LIN {X 0,Y 354.801,Z 259.294,A -85,B 0,C 180,E1 -13349.685,E2 -13349.685} C_VEL
LIN {X 0,Y 354.812,Z 259.29,A -85,B 0,C 180,E1 -13353.685,E2 -13353.685} C_VEL
LIN {X 0,Y 354.795,Z 259.291,A -85,B 0,C 180,E1 -13356.461,E2 -13356.461} C_VEL
LIN {X 0,Y 354.823,Z 259.288,A -85,B 0,C 180,E1 -13359.425,E2 -13359.425} C_VEL
LIN {X 0,Y 354.787,Z 259.29,A -85,B 0,C 180,E1 -13362.869,E2 -13362.869} C_VEL
LIN {X 0,Y 354.791,Z 259.41,A -85,B 0,C 180,E1 -13364.212,E2 -13364.212} C_VEL
LIN {X 0,Y 355.557,Z 263.624,A -85,B 0,C 180,E1 -13367.776,E2 -13367.776} C_VEL
LIN {X 0,Y 356.179,Z 267.564,A -85,B 0,C 180,E1 -13370.847,E2 -13370.847} C_VEL
LIN {X 0,Y 356.609,Z 271.764,A -85,B 0,C 180,E1 -13373.905,E2 -13373.905} C_VEL
LIN {X 0,Y 356.289,Z 275.58,A -85,B 0,C 180,E1 -13376.475,E2 -13376.475} C_VEL
LIN {X 0,Y 355.724,Z 280.665,A -85,B 0,C 180,E1 -13379.749,E2 -13379.749} C_VEL
LIN {X 0,Y 355.068,Z 285.864,A -85,B 0,C 180,E1 -13382.964,E2 -13382.964} C_VEL
LIN {X 0,Y 354.552,Z 291.984,A -85,B 0,C 180,E1 -13386.645,E2 -13386.645} C_VEL
LIN {X 0,Y 354.356,Z 295.247,A -85,B 0,C 180,E1 -13388.455,E2 -13388.455} C_VEL
LIN {X 0,Y 357.769,Z 308.674,A -85,B 0,C 180,E1 -13389.219,E2 -13389.219} C_VEL
LIN {X 0,Y 360.089,Z 320.881,A -85,B 0,C 180,E1 -13390.079,E2 -13390.079} C_VEL
LIN {X 0,Y 361.243,Z 331.83,A -85,B 0,C 180,E1 -13390.982,E2 -13390.982} C_VEL
LIN {X 0,Y 360.677,Z 339.868,A -85,B 0,C 180,E1 -13391.688,E2 -13391.688} C_VEL
LIN {X 0,Y 359.136,Z 351.571,A -85,B 0,C 180,E1 -13392.931,E2 -13392.931} C_VEL
LIN {X 0,Y 357.813,Z 361.437,A -85,B 0,C 180,E1 -13394.249,E2 -13394.249} C_VEL
LIN {X 0,Y 356.726,Z 370.441,A -85,B 0,C 180,E1 -13395.744,E2 -13395.744} C_VEL
LIN {X 0,Y 355.47,Z 378.705,A -85,B 0,C 180,E1 -13397.439,E2 -13397.439} C_VEL
LIN {X 0,Y 354.633,Z 385.385,A -85,B 0,C 180,E1 -13399.149,E2 -13399.149} C_VEL
LIN {X 0,Y 353.992,Z 390.739,A -85,B 0,C 180,E1 -13400.861,E2 -13400.861} C_VEL
LIN {X 0,Y 353.547,Z 394.934,A -85,B 0,C 180,E1 -13402.576,E2 -13402.576} C_VEL
LIN {X 0,Y 353.314,Z 398.087,A -85,B 0,C 180,E1 -13404.292,E2 -13404.292} C_VEL
LIN {X 0,Y 353.266,Z 399.668,A -85,B 0,C 180,E1 -13405.436,E2 -13405.436} C_VEL
LIN {X 0,Y 353.22,Z 400.829,A -85,B 0,C 180,E1 -13406.578,E2 -13406.578} C_VEL
LIN {X 0,Y 353.204,Z 401.911,A -85,B 0,C 180,E1 -13408.86,E2 -13408.86} C_VEL
LIN {X 0,Y 353.264,Z 401.877,A -85,B 0,C 180,E1 -13410,E2 -13410} C_VEL
LIN {X 0,Y 353.223,Z 401.444,A -85,B 0,C 180,E1 -13411.14,E2 -13411.14} C_VEL
LIN {X 0,Y 353.226,Z 399.304,A -85,B 0,C 180,E1 -13413.422,E2 -13413.422} C_VEL
LIN {X 0,Y 353.258,Z 396.601,A -85,B 0,C 180,E1 -13415.136,E2 -13415.136} C_VEL
LIN {X 0,Y 353.419,Z 392.866,A -85,B 0,C 180,E1 -13416.852,E2 -13416.852} C_VEL
LIN {X 0,Y 353.702,Z 387.997,A -85,B 0,C 180,E1 -13418.57,E2 -13418.57} C_VEL
LIN {X 0,Y 354.198,Z 381.846,A -85,B 0,C 180,E1 -13420.287,E2 -13420.287} C_VEL
LIN {X 0,Y 354.851,Z 374.184,A -85,B 0,C 180,E1 -13422.002,E2 -13422.002} C_VEL
LIN {X 0,Y 355.604,Z 366.332,A -85,B 0,C 180,E1 -13423.428,E2 -13423.428} C_VEL
LIN {X 0,Y 356.485,Z 356.718,A -85,B 0,C 180,E1 -13424.85,E2 -13424.85} C_VEL
LIN {X 0,Y 357.37,Z 346.037,A -85,B 0,C 180,E1 -13426.127,E2 -13426.127} C_VEL
LIN {X 0,Y 358.522,Z 334.094,A -85,B 0,C 180,E1 -13427.247,E2 -13427.247} C_VEL
LIN {X 0,Y 358.749,Z 330.526,A -85,B 0,C 180,E1 -13427.529,E2 -13427.529} C_VEL
LIN {X 0,Y 357.34,Z 318.321,A -85,B 0,C 180,E1 -13428.423,E2 -13428.423} C_VEL
LIN {X 0,Y 355.4,Z 304.853,A -85,B 0,C 180,E1 -13429.164,E2 -13429.164} C_VEL
LIN {X 0,Y 353.852,Z 295.492,A -85,B 0,C 180,E1 -13429.544,E2 -13429.544} C_VEL
LIN {X 0,Y 354.18,Z 289.708,A -85,B 0,C 180,E1 -13432.764,E2 -13432.764} C_VEL
LIN {X 0,Y 354.551,Z 284.261,A -85,B 0,C 180,E1 -13435.854,E2 -13435.854} C_VEL
LIN {X 0,Y 355.08,Z 277.706,A -85,B 0,C 180,E1 -13439.657,E2 -13439.657} C_VEL
LIN {X 0,Y 355.598,Z 272.227,A -85,B 0,C 180,E1 -13442.922,E2 -13442.922} C_VEL
LIN {X 0,Y 355.985,Z 267.281,A -85,B 0,C 180,E1 -13445.957,E2 -13445.957} C_VEL
LIN {X 0,Y 355.526,Z 263.384,A -85,B 0,C 180,E1 -13448.511,E2 -13448.511} C_VEL
LIN {X 0,Y 354.84,Z 259.286,A -85,B 0,C 180,E1 -13451.394,E2 -13451.394} C_VEL
LIN {X 0,Y 354.743,Z 259.295,A -85,B 0,C 180,E1 -13455.496,E2 -13455.496} C_VEL
LIN {X 0,Y 354.76,Z 259.294,A -85,B 0,C 180,E1 -13459.174,E2 -13459.174} C_VEL
LIN {X 0,Y 354.796,Z 259.29,A -85,B 0,C 180,E1 -13462.403,E2 -13462.403} C_VEL
LIN {X 0,Y 354.805,Z 259.29,A -85,B 0,C 180,E1 -13464.939,E2 -13464.939} C_VEL
LIN {X 0,Y 354.79,Z 259.292,A -85,B 0,C 180,E1 -13468.404,E2 -13468.404} C_VEL
LIN {X 0,Y 354.796,Z 259.287,A -85,B 0,C 180,E1 -13471.613,E2 -13471.613} C_VEL
LIN {X 0,Y 354.83,Z 259.283,A -85,B 0,C 180,E1 -13475.656,E2 -13475.656} C_VEL
LIN {X 0,Y 354.821,Z 259.285,A -85,B 0,C 180,E1 -13479.112,E2 -13479.112} C_VEL
LIN {X 0,Y 354.893,Z 259.277,A -85,B 0,C 180,E1 -13482.718,E2 -13482.718} C_VEL
LIN {X 0,Y 354.946,Z 259.274,A -85,B 0,C 180,E1 -13486.254,E2 -13486.254} C_VEL
LIN {X 0,Y 354.971,Z 259.268,A -85,B 0,C 180,E1 -13489.734,E2 -13489.734} C_VEL
LIN {X 0,Y 355.119,Z 259.247,A -85,B 0,C 180,E1 -13493.179,E2 -13493.179} C_VEL
LIN {X 0,Y 355.237,Z 259.236,A -85,B 0,C 180,E1 -13497.731,E2 -13497.731} C_VEL
LIN {X 0,Y 355.391,Z 259.218,A -85,B 0,C 180,E1 -13499.999,E2 -13499.999} C_VEL
LIN {X 0,Y 355.238,Z 259.234,A -85,B 0,C 180,E1 -13502.266,E2 -13502.266} C_VEL
LIN {X 0,Y 355.13,Z 259.246,A -85,B 0,C 180,E1 -13506.818,E2 -13506.818} C_VEL
LIN {X 0,Y 355.007,Z 259.262,A -85,B 0,C 180,E1 -13509.111,E2 -13509.111} C_VEL
LIN {X 0,Y 354.912,Z 259.273,A -85,B 0,C 180,E1 -13512.58,E2 -13512.58} C_VEL
LIN {X 0,Y 354.879,Z 259.278,A -85,B 0,C 180,E1 -13516.095,E2 -13516.095} C_VEL
LIN {X 0,Y 354.891,Z 259.275,A -85,B 0,C 180,E1 -13518.471,E2 -13518.471} C_VEL
LIN {X 0,Y 354.824,Z 259.284,A -85,B 0,C 180,E1 -13522.105,E2 -13522.105} C_VEL
LIN {X 0,Y 354.889,Z 259.277,A -85,B 0,C 180,E1 -13525.826,E2 -13525.826} C_VEL
LIN {X 0,Y 354.844,Z 259.283,A -85,B 0,C 180,E1 -13529.678,E2 -13529.678} C_VEL
LIN {X 0,Y 354.795,Z 259.288,A -85,B 0,C 180,E1 -13533.701,E2 -13533.701} C_VEL
LIN {X 0,Y 354.788,Z 259.289,A -85,B 0,C 180,E1 -13536.459,E2 -13536.459} C_VEL
LIN {X 0,Y 354.813,Z 259.287,A -85,B 0,C 180,E1 -13539.423,E2 -13539.423} C_VEL
LIN {X 0,Y 354.823,Z 259.29,A -85,B 0,C 180,E1 -13542.875,E2 -13542.875} C_VEL
LIN {X 0,Y 354.773,Z 259.29,A -85,B 0,C 180,E1 -13546.106,E2 -13546.106} C_VEL
LIN {X 0,Y 354.777,Z 259.291,A -85,B 0,C 180,E1 -13549.179,E2 -13549.179} C_VEL
LIN {X 0,Y 354.8,Z 259.29,A -85,B 0,C 180,E1 -13552.401,E2 -13552.401} C_VEL
LIN {X 0,Y 354.8,Z 259.289,A -85,B 0,C 180,E1 -13554.94,E2 -13554.94} C_VEL
LIN {X 0,Y 354.782,Z 259.294,A -85,B 0,C 180,E1 -13558.405,E2 -13558.405} C_VEL
LIN {X 0,Y 354.825,Z 259.284,A -85,B 0,C 180,E1 -13561.617,E2 -13561.617} C_VEL
LIN {X 0,Y 354.816,Z 259.288,A -85,B 0,C 180,E1 -13564.167,E2 -13564.167} C_VEL
LIN {X 0,Y 354.703,Z 259.301,A -85,B 0,C 180,E1 -13566.655,E2 -13566.655} C_VEL
LIN {X 0,Y 354.621,Z 259.436,A -85,B 0,C 180,E1 -13568.344,E2 -13568.344} C_VEL
LIN {X 0,Y 354.458,Z 263.774,A -85,B 0,C 180,E1 -13572.117,E2 -13572.117} C_VEL
LIN {X 0,Y 354.257,Z 268.889,A -85,B 0,C 180,E1 -13576.425,E2 -13576.425} C_VEL
LIN {X 0,Y 354.011,Z 274.308,A -85,B 0,C 180,E1 -13580.862,E2 -13580.862} C_VEL
LIN {X 0,Y 354.001,Z 277.677,A -85,B 0,C 180,E1 -13583.549,E2 -13583.549} C_VEL
LIN {X 0,Y 356.74,Z 290.857,A -85,B 0,C 180,E1 -13584.182,E2 -13584.182} C_VEL
LIN {X 0,Y 358.805,Z 303.884,A -85,B 0,C 180,E1 -13585.014,E2 -13585.014} C_VEL
LIN {X 0,Y 359.321,Z 308.615,A -85,B 0,C 180,E1 -13585.372,E2 -13585.372} C_VEL
LIN {X 0,Y 358.466,Z 320.435,A -85,B 0,C 180,E1 -13586.347,E2 -13586.347} C_VEL
LIN {X 0,Y 357.382,Z 332.207,A -85,B 0,C 180,E1 -13587.605,E2 -13587.605} C_VEL
LIN {X 0,Y 356.509,Z 341.682,A -85,B 0,C 180,E1 -13588.87,E2 -13588.87} C_VEL
LIN {X 0,Y 355.705,Z 350.333,A -85,B 0,C 180,E1 -13590.283,E2 -13590.283} C_VEL
LIN {X 0,Y 354.784,Z 358.758,A -85,B 0,C 180,E1 -13591.987,E2 -13591.987} C_VEL
LIN {X 0,Y 354.232,Z 365.515,A -85,B 0,C 180,E1 -13593.697,E2 -13593.697} C_VEL
LIN {X 0,Y 353.784,Z 371.732,A -85,B 0,C 180,E1 -13595.7,E2 -13595.7} C_VEL
LIN {X 0,Y 353.482,Z 375.785,A -85,B 0,C 180,E1 -13597.425,E2 -13597.425} C_VEL
LIN {X 0,Y 353.222,Z 378.791,A -85,B 0,C 180,E1 -13599.159,E2 -13599.159} C_VEL
LIN {X 0,Y 353.115,Z 380.238,A -85,B 0,C 180,E1 -13600.319,E2 -13600.319} C_VEL
LIN {X 0,Y 353.117,Z 381.259,A -85,B 0,C 180,E1 -13601.48,E2 -13601.48} C_VEL
LIN {X 0,Y 353.144,Z 381.957,A -85,B 0,C 180,E1 -13602.806,E2 -13602.806} C_VEL
LIN {X 0,Y 353.098,Z 381.895,A -85,B 0,C 180,E1 -13604.995,E2 -13604.995} C_VEL
LIN {X 0,Y 353.224,Z 381.265,A -85,B 0,C 180,E1 -13606.173,E2 -13606.173} C_VEL
LIN {X 0,Y 353.36,Z 380.231,A -85,B 0,C 180,E1 -13607.357,E2 -13607.357} C_VEL
LIN {X 0,Y 353.527,Z 378.734,A -85,B 0,C 180,E1 -13608.546,E2 -13608.546} C_VEL
LIN {X 0,Y 353.964,Z 375.623,A -85,B 0,C 180,E1 -13610.332,E2 -13610.332} C_VEL
LIN {X 0,Y 354.54,Z 371.367,A -85,B 0,C 180,E1 -13612.125,E2 -13612.125} C_VEL
LIN {X 0,Y 355.463,Z 364.784,A -85,B 0,C 180,E1 -13614.22,E2 -13614.22} C_VEL
LIN {X 0,Y 356.534,Z 357.492,A -85,B 0,C 180,E1 -13616.013,E2 -13616.013} C_VEL
LIN {X 0,Y 357.608,Z 350.251,A -85,B 0,C 180,E1 -13617.452,E2 -13617.452} C_VEL
LIN {X 0,Y 358.904,Z 340.748,A -85,B 0,C 180,E1 -13618.989,E2 -13618.989} C_VEL
LIN {X 0,Y 360.219,Z 330.531,A -85,B 0,C 180,E1 -13620.319,E2 -13620.319} C_VEL
LIN {X 0,Y 361.445,Z 319.694,A -85,B 0,C 180,E1 -13621.443,E2 -13621.443} C_VEL
LIN {X 0,Y 362.367,Z 310.873,A -85,B 0,C 180,E1 -13622.179,E2 -13622.179} C_VEL
LIN {X 0,Y 360.465,Z 300.228,A -85,B 0,C 180,E1 -13623.086,E2 -13623.086} C_VEL
LIN {X 0,Y 356.959,Z 287.408,A -85,B 0,C 180,E1 -13624.031,E2 -13624.031} C_VEL
LIN {X 0,Y 354.026,Z 278.062,A -85,B 0,C 180,E1 -13624.629,E2 -13624.629} C_VEL
LIN {X 0,Y 354.261,Z 274.211,A -85,B 0,C 180,E1 -13627.95,E2 -13627.95} C_VEL
LIN {X 0,Y 354.295,Z 273.377,A -85,B 0,C 180,E1 -13628.691,E2 -13628.691} C_VEL
LIN {X 0,Y 353.72,Z 272.417,A -85,B 0,C 180,E1 -13629.629,E2 -13629.629} C_VEL
LIN {X 0,Y 351.022,Z 271.112,A -85,B 0,C 180,E1 -13631.165,E2 -13631.165} C_VEL
LIN {X 0,Y 348.724,Z 270.103,A -85,B 0,C 180,E1 -13632.409,E2 -13632.409} C_VEL
LIN {X 0,Y 347.77,Z 269.229,A -85,B 0,C 180,E1 -13633.367,E2 -13633.367} C_VEL
LIN {X 0,Y 347.711,Z 268.9,A -85,B 0,C 180,E1 -13633.689,E2 -13633.689} C_VEL
LIN {X 0,Y 347.998,Z 265.854,A -85,B 0,C 180,E1 -13636.637,E2 -13636.637} C_VEL
LIN {X 0,Y 348.017,Z 262.805,A -85,B 0,C 180,E1 -13639.745,E2 -13639.745} C_VEL
LIN {X 0,Y 347.754,Z 260.169,A -85,B 0,C 180,E1 -13642.68,E2 -13642.68} C_VEL
LIN {X 0,Y 347.737,Z 260.175,A -85,B 0,C 180,E1 -13645.957,E2 -13645.957} C_VEL
LIN {X 0,Y 347.753,Z 260.169,A -85,B 0,C 180,E1 -13649.654,E2 -13649.654} C_VEL
LIN {X 0,Y 347.841,Z 260.156,A -85,B 0,C 180,E1 -13652.745,E2 -13652.745} C_VEL
LIN {X 0,Y 347.789,Z 260.166,A -85,B 0,C 180,E1 -13656.164,E2 -13656.164} C_VEL
LIN {X 0,Y 347.826,Z 260.157,A -85,B 0,C 180,E1 -13659.912,E2 -13659.912} C_VEL
LIN {X 0,Y 347.857,Z 260.152,A -85,B 0,C 180,E1 -13662.36,E2 -13662.36} C_VEL
LIN {X 0,Y 347.888,Z 260.149,A -85,B 0,C 180,E1 -13665.972,E2 -13665.972} C_VEL
LIN {X 0,Y 347.919,Z 260.148,A -85,B 0,C 180,E1 -13669.527,E2 -13669.527} C_VEL
LIN {X 0,Y 348.082,Z 260.128,A -85,B 0,C 180,E1 -13673.043,E2 -13673.043} C_VEL
LIN {X 0,Y 348.2,Z 260.112,A -85,B 0,C 180,E1 -13677.688,E2 -13677.688} C_VEL
LIN {X 0,Y 348.315,Z 260.096,A -85,B 0,C 180,E1 -13680.001,E2 -13680.001} C_VEL
LIN {X 0,Y 348.2,Z 260.113,A -85,B 0,C 180,E1 -13682.315,E2 -13682.315} C_VEL
LIN {X 0,Y 348.097,Z 260.125,A -85,B 0,C 180,E1 -13686.959,E2 -13686.959} C_VEL
LIN {X 0,Y 347.922,Z 260.147,A -85,B 0,C 180,E1 -13690.476,E2 -13690.476} C_VEL
LIN {X 0,Y 347.893,Z 260.153,A -85,B 0,C 180,E1 -13694.151,E2 -13694.151} C_VEL
LIN {X 0,Y 347.887,Z 260.155,A -85,B 0,C 180,E1 -13698.292,E2 -13698.292} C_VEL
LIN {X 0,Y 347.784,Z 260.17,A -85,B 0,C 180,E1 -13701.636,E2 -13701.636} C_VEL
LIN {X 0,Y 347.795,Z 260.168,A -85,B 0,C 180,E1 -13705.111,E2 -13705.111} C_VEL
LIN {X 0,Y 347.756,Z 260.172,A -85,B 0,C 180,E1 -13707.7,E2 -13707.7} C_VEL
LIN {X 0,Y 347.738,Z 260.174,A -85,B 0,C 180,E1 -13710.35,E2 -13710.35} C_VEL
LIN {X 0,Y 347.746,Z 260.171,A -85,B 0,C 180,E1 -13714.045,E2 -13714.045} C_VEL
LIN {X 0,Y 347.759,Z 260.167,A -85,B 0,C 180,E1 -13717.322,E2 -13717.322} C_VEL
LIN {X 0,Y 347.731,Z 260.165,A -85,B 0,C 180,E1 -13720.299,E2 -13720.299} C_VEL
LIN {X 0,Y 347.729,Z 260.194,A -85,B 0,C 180,E1 -13723.608,E2 -13723.608} C_VEL
LIN {X 0,Y 348.362,Z 263.721,A -85,B 0,C 180,E1 -13726.693,E2 -13726.693} C_VEL
LIN {X 0,Y 349.028,Z 267.661,A -85,B 0,C 180,E1 -13729.923,E2 -13729.923} C_VEL
LIN {X 0,Y 349.554,Z 271.573,A -85,B 0,C 180,E1 -13732.904,E2 -13732.904} C_VEL
LIN {X 0,Y 349.45,Z 275.595,A -85,B 0,C 180,E1 -13735.729,E2 -13735.729} C_VEL
LIN {X 0,Y 348.692,Z 281.673,A -85,B 0,C 180,E1 -13739.744,E2 -13739.744} C_VEL
LIN {X 0,Y 347.895,Z 287.826,A -85,B 0,C 180,E1 -13743.614,E2 -13743.614} C_VEL
LIN {X 0,Y 347.477,Z 292.973,A -85,B 0,C 180,E1 -13746.772,E2 -13746.772} C_VEL
LIN {X 0,Y 347.353,Z 294.823,A -85,B 0,C 180,E1 -13747.889,E2 -13747.889} C_VEL
LIN {X 0,Y 350.974,Z 309.105,A -85,B 0,C 180,E1 -13748.744,E2 -13748.744} C_VEL
LIN {X 0,Y 353.166,Z 320.098,A -85,B 0,C 180,E1 -13749.547,E2 -13749.547} C_VEL
LIN {X 0,Y 354.42,Z 330.812,A -85,B 0,C 180,E1 -13750.451,E2 -13750.451} C_VEL
LIN {X 0,Y 354.501,Z 335.805,A -85,B 0,C 180,E1 -13750.907,E2 -13750.907} C_VEL
LIN {X 0,Y 353.103,Z 347.135,A -85,B 0,C 180,E1 -13752.031,E2 -13752.031} C_VEL
LIN {X 0,Y 351.582,Z 357.393,A -85,B 0,C 180,E1 -13753.301,E2 -13753.301} C_VEL
LIN {X 0,Y 350.502,Z 365.948,A -85,B 0,C 180,E1 -13754.621,E2 -13754.621} C_VEL
LIN {X 0,Y 349.196,Z 374.926,A -85,B 0,C 180,E1 -13756.321,E2 -13756.321} C_VEL
LIN {X 0,Y 348.021,Z 382.301,A -85,B 0,C 180,E1 -13758.054,E2 -13758.054} C_VEL
LIN {X 0,Y 347.144,Z 389.122,A -85,B 0,C 180,E1 -13760.091,E2 -13760.091} C_VEL
LIN {X 0,Y 346.647,Z 393.641,A -85,B 0,C 180,E1 -13761.841,E2 -13761.841} C_VEL
LIN {X 0,Y 346.246,Z 397.795,A -85,B 0,C 180,E1 -13764.044,E2 -13764.044} C_VEL
LIN {X 0,Y 346.166,Z 399.556,A -85,B 0,C 180,E1 -13765.342,E2 -13765.342} C_VEL
LIN {X 0,Y 346.143,Z 400.678,A -85,B 0,C 180,E1 -13766.508,E2 -13766.508} C_VEL
LIN {X 0,Y 346.105,Z 401.72,A -85,B 0,C 180,E1 -13768.837,E2 -13768.837} C_VEL
LIN {X 0,Y 346.166,Z 401.667,A -85,B 0,C 180,E1 -13770,E2 -13770} C_VEL
LIN {X 0,Y 346.124,Z 401.198,A -85,B 0,C 180,E1 -13771.163,E2 -13771.163} C_VEL
LIN {X 0,Y 346.15,Z 399.018,A -85,B 0,C 180,E1 -13773.492,E2 -13773.492} C_VEL
LIN {X 0,Y 346.189,Z 395.828,A -85,B 0,C 180,E1 -13775.483,E2 -13775.483} C_VEL
LIN {X 0,Y 346.44,Z 390.998,A -85,B 0,C 180,E1 -13777.577,E2 -13777.577} C_VEL
LIN {X 0,Y 346.861,Z 384.643,A -85,B 0,C 180,E1 -13779.623,E2 -13779.623} C_VEL
LIN {X 0,Y 347.423,Z 377.709,A -85,B 0,C 180,E1 -13781.375,E2 -13781.375} C_VEL
LIN {X 0,Y 348.379,Z 369.03,A -85,B 0,C 180,E1 -13783.117,E2 -13783.117} C_VEL
LIN {X 0,Y 349.301,Z 358.868,A -85,B 0,C 180,E1 -13784.752,E2 -13784.752} C_VEL
LIN {X 0,Y 350.15,Z 349.327,A -85,B 0,C 180,E1 -13785.99,E2 -13785.99} C_VEL
LIN {X 0,Y 351.042,Z 339.51,A -85,B 0,C 180,E1 -13787.025,E2 -13787.025} C_VEL
LIN {X 0,Y 351.795,Z 331.299,A -85,B 0,C 180,E1 -13787.73,E2 -13787.73} C_VEL
LIN {X 0,Y 350.483,Z 319.676,A -85,B 0,C 180,E1 -13788.625,E2 -13788.625} C_VEL
LIN {X 0,Y 348.643,Z 306.367,A -85,B 0,C 180,E1 -13789.404,E2 -13789.404} C_VEL
LIN {X 0,Y 346.777,Z 295.257,A -85,B 0,C 180,E1 -13789.882,E2 -13789.882} C_VEL
LIN {X 0,Y 347.155,Z 289.384,A -85,B 0,C 180,E1 -13793.251,E2 -13793.251} C_VEL
LIN {X 0,Y 347.668,Z 282.622,A -85,B 0,C 180,E1 -13797.194,E2 -13797.194} C_VEL
LIN {X 0,Y 348.239,Z 276.307,A -85,B 0,C 180,E1 -13800.972,E2 -13800.972} C_VEL
LIN {X 0,Y 348.803,Z 270.824,A -85,B 0,C 180,E1 -13804.344,E2 -13804.344} C_VEL
LIN {X 0,Y 348.947,Z 267.706,A -85,B 0,C 180,E1 -13806.328,E2 -13806.328} C_VEL
LIN {X 0,Y 348.458,Z 264.187,A -85,B 0,C 180,E1 -13808.698,E2 -13808.698} C_VEL
LIN {X 0,Y 347.785,Z 260.165,A -85,B 0,C 180,E1 -13811.608,E2 -13811.608} C_VEL
LIN {X 0,Y 347.69,Z 260.177,A -85,B 0,C 180,E1 -13815.028,E2 -13815.028} C_VEL
LIN {X 0,Y 347.704,Z 260.172,A -85,B 0,C 180,E1 -13818.404,E2 -13818.404} C_VEL
LIN {X 0,Y 347.759,Z 260.164,A -85,B 0,C 180,E1 -13822.013,E2 -13822.013} C_VEL
LIN {X 0,Y 347.74,Z 260.166,A -85,B 0,C 180,E1 -13825.534,E2 -13825.534} C_VEL
LIN {X 0,Y 347.742,Z 260.168,A -85,B 0,C 180,E1 -13828.299,E2 -13828.299} C_VEL
LIN {X 0,Y 347.742,Z 260.168,A -85,B 0,C 180,E1 -13830.983,E2 -13830.983} C_VEL
LIN {X 0,Y 347.744,Z 260.165,A -85,B 0,C 180,E1 -13833.599,E2 -13833.599} C_VEL
LIN {X 0,Y 347.762,Z 260.166,A -85,B 0,C 180,E1 -13836.159,E2 -13836.159} C_VEL
LIN {X 0,Y 347.8,Z 260.16,A -85,B 0,C 180,E1 -13839.907,E2 -13839.907} C_VEL
LIN {X 0,Y 347.861,Z 260.156,A -85,B 0,C 180,E1 -13842.358,E2 -13842.358} C_VEL
LIN {X 0,Y 347.893,Z 260.15,A -85,B 0,C 180,E1 -13845.969,E2 -13845.969} C_VEL
LIN {X 0,Y 347.922,Z 260.144,A -85,B 0,C 180,E1 -13849.524,E2 -13849.524} C_VEL
LIN {X 0,Y 348.085,Z 260.123,A -85,B 0,C 180,E1 -13853.041,E2 -13853.041} C_VEL
LIN {X 0,Y 348.2,Z 260.112,A -85,B 0,C 180,E1 -13857.685,E2 -13857.685} C_VEL
LIN {X 0,Y 348.361,Z 260.094,A -85,B 0,C 180,E1 -13859.999,E2 -13859.999} C_VEL
LIN {X 0,Y 348.201,Z 260.11,A -85,B 0,C 180,E1 -13862.312,E2 -13862.312} C_VEL
LIN {X 0,Y 348.098,Z 260.122,A -85,B 0,C 180,E1 -13866.956,E2 -13866.956} C_VEL
LIN {X 0,Y 347.959,Z 260.141,A -85,B 0,C 180,E1 -13869.297,E2 -13869.297} C_VEL
LIN {X 0,Y 347.881,Z 260.149,A -85,B 0,C 180,E1 -13872.838,E2 -13872.838} C_VEL
LIN {X 0,Y 347.829,Z 260.155,A -85,B 0,C 180,E1 -13876.43,E2 -13876.43} C_VEL
LIN {X 0,Y 347.841,Z 260.154,A -85,B 0,C 180,E1 -13878.859,E2 -13878.859} C_VEL
LIN {X 0,Y 347.764,Z 260.163,A -85,B 0,C 180,E1 -13882.578,E2 -13882.578} C_VEL
LIN {X 0,Y 347.802,Z 260.162,A -85,B 0,C 180,E1 -13885.107,E2 -13885.107} C_VEL
LIN {X 0,Y 347.802,Z 260.16,A -85,B 0,C 180,E1 -13887.693,E2 -13887.693} C_VEL
LIN {X 0,Y 347.754,Z 260.164,A -85,B 0,C 180,E1 -13890.346,E2 -13890.346} C_VEL
LIN {X 0,Y 347.733,Z 260.168,A -85,B 0,C 180,E1 -13894.463,E2 -13894.463} C_VEL
LIN {X 0,Y 347.765,Z 260.163,A -85,B 0,C 180,E1 -13897.988,E2 -13897.988} C_VEL
LIN {X 0,Y 347.773,Z 260.162,A -85,B 0,C 180,E1 -13901.608,E2 -13901.608} C_VEL
LIN {X 0,Y 347.785,Z 260.164,A -85,B 0,C 180,E1 -13905.011,E2 -13905.011} C_VEL
LIN {X 0,Y 347.739,Z 260.168,A -85,B 0,C 180,E1 -13908.397,E2 -13908.397} C_VEL
LIN {X 0,Y 347.765,Z 260.163,A -85,B 0,C 180,E1 -13912.01,E2 -13912.01} C_VEL
LIN {X 0,Y 347.733,Z 260.167,A -85,B 0,C 180,E1 -13915.536,E2 -13915.536} C_VEL
LIN {X 0,Y 347.733,Z 260.17,A -85,B 0,C 180,E1 -13918.3,E2 -13918.3} C_VEL
LIN {X 0,Y 347.763,Z 260.164,A -85,B 0,C 180,E1 -13920.987,E2 -13920.987} C_VEL
LIN {X 0,Y 347.775,Z 260.162,A -85,B 0,C 180,E1 -13923.604,E2 -13923.604} C_VEL
LIN {X 0,Y 347.686,Z 260.177,A -85,B 0,C 180,E1 -13926.155,E2 -13926.155} C_VEL
LIN {X 0,Y 347.579,Z 260.275,A -85,B 0,C 180,E1 -13928.297,E2 -13928.297} C_VEL
LIN {X 0,Y 347.387,Z 264.853,A -85,B 0,C 180,E1 -13932.334,E2 -13932.334} C_VEL
LIN {X 0,Y 347.194,Z 269.486,A -85,B 0,C 180,E1 -13936.311,E2 -13936.311} C_VEL
LIN {X 0,Y 346.957,Z 274.754,A -85,B 0,C 180,E1 -13940.674,E2 -13940.674} C_VEL
LIN {X 0,Y 346.953,Z 277.847,A -85,B 0,C 180,E1 -13943.211,E2 -13943.211} C_VEL
LIN {X 0,Y 349.868,Z 291.864,A -85,B 0,C 180,E1 -13943.914,E2 -13943.914} C_VEL
LIN {X 0,Y 351.753,Z 303.801,A -85,B 0,C 180,E1 -13944.698,E2 -13944.698} C_VEL
LIN {X 0,Y 352.418,Z 309.462,A -85,B 0,C 180,E1 -13945.138,E2 -13945.138} C_VEL
LIN {X 0,Y 351.521,Z 321.106,A -85,B 0,C 180,E1 -13946.131,E2 -13946.131} C_VEL
LIN {X 0,Y 350.421,Z 332.79,A -85,B 0,C 180,E1 -13947.414,E2 -13947.414} C_VEL
LIN {X 0,Y 349.646,Z 341.22,A -85,B 0,C 180,E1 -13948.56,E2 -13948.56} C_VEL
LIN {X 0,Y 348.756,Z 349.989,A -85,B 0,C 180,E1 -13950,E2 -13950} C_VEL
LIN {X 0,Y 347.79,Z 358.545,A -85,B 0,C 180,E1 -13951.737,E2 -13951.737} C_VEL
LIN {X 0,Y 347.216,Z 365.376,A -85,B 0,C 180,E1 -13953.481,E2 -13953.481} C_VEL
LIN {X 0,Y 346.773,Z 370.853,A -85,B 0,C 180,E1 -13955.233,E2 -13955.233} C_VEL
LIN {X 0,Y 346.473,Z 375.149,A -85,B 0,C 180,E1 -13956.99,E2 -13956.99} C_VEL
LIN {X 0,Y 346.286,Z 377.434,A -85,B 0,C 180,E1 -13958.167,E2 -13958.167} C_VEL
LIN {X 0,Y 346.114,Z 379.258,A -85,B 0,C 180,E1 -13959.348,E2 -13959.348} C_VEL
LIN {X 0,Y 346.022,Z 380.628,A -85,B 0,C 180,E1 -13960.532,E2 -13960.532} C_VEL
LIN {X 0,Y 346.015,Z 381.597,A -85,B 0,C 180,E1 -13961.719,E2 -13961.719} C_VEL
LIN {X 0,Y 346.04,Z 382.17,A -85,B 0,C 180,E1 -13962.909,E2 -13962.909} C_VEL
LIN {X 0,Y 346.016,Z 382.298,A -85,B 0,C 180,E1 -13964.107,E2 -13964.107} C_VEL
LIN {X 0,Y 346.023,Z 382.016,A -85,B 0,C 180,E1 -13965.31,E2 -13965.31} C_VEL
LIN {X 0,Y 346.299,Z 380.467,A -85,B 0,C 180,E1 -13967.482,E2 -13967.482} C_VEL
LIN {X 0,Y 346.664,Z 377.696,A -85,B 0,C 180,E1 -13969.542,E2 -13969.542} C_VEL
LIN {X 0,Y 347.204,Z 374.023,A -85,B 0,C 180,E1 -13971.395,E2 -13971.395} C_VEL
LIN {X 0,Y 347.902,Z 369.279,A -85,B 0,C 180,E1 -13973.198,E2 -13973.198} C_VEL
LIN {X 0,Y 348.825,Z 363.105,A -85,B 0,C 180,E1 -13975.03,E2 -13975.03} C_VEL
LIN {X 0,Y 350.078,Z 355.343,A -85,B 0,C 180,E1 -13976.852,E2 -13976.852} C_VEL
LIN {X 0,Y 351.407,Z 346.532,A -85,B 0,C 180,E1 -13978.5,E2 -13978.5} C_VEL
LIN {X 0,Y 352.856,Z 336.301,A -85,B 0,C 180,E1 -13980.027,E2 -13980.027} C_VEL
LIN {X 0,Y 354.254,Z 325.306,A -85,B 0,C 180,E1 -13981.337,E2 -13981.337} C_VEL
LIN {X 0,Y 355.552,Z 314.193,A -85,B 0,C 180,E1 -13982.368,E2 -13982.368} C_VEL
LIN {X 0,Y 355.495,Z 310.232,A -85,B 0,C 180,E1 -13982.717,E2 -13982.717} C_VEL
LIN {X 0,Y 353.432,Z 299.879,A -85,B 0,C 180,E1 -13983.628,E2 -13983.628} C_VEL
LIN {X 0,Y 349.936,Z 287.394,A -85,B 0,C 180,E1 -13984.573,E2 -13984.573} C_VEL
LIN {X 0,Y 347.076,Z 278.671,A -85,B 0,C 180,E1 -13985.139,E2 -13985.139} C_VEL
LIN {X 0,Y 347.032,Z 278.243,A -85,B 0,C 180,E1 -13985.197,E2 -13985.197} C_VEL
LIN {X 0,Y 347.29,Z 274.125,A -85,B 0,C 180,E1 -13988.853,E2 -13988.853} C_VEL
LIN {X 0,Y 347.54,Z 270.843,A -85,B 0,C 180,E1 -13991.86,E2 -13991.86} C_VEL
LIN {X 0,Y 347.711,Z 268.9,A -85,B 0,C 180,E1 -13993.689,E2 -13993.689} C_VEL
LIN {X 0,Y 347.132,Z 267.994,A -85,B 0,C 180,E1 -13994.646,E2 -13994.646} C_VEL
LIN {X 0,Y 344.456,Z 266.816,A -85,B 0,C 180,E1 -13996.215,E2 -13996.215} C_VEL
LIN {X 0,Y 342.144,Z 265.926,A -85,B 0,C 180,E1 -13997.486,E2 -13997.486} C_VEL
LIN {X 0,Y 341.129,Z 265.145,A -85,B 0,C 180,E1 -13998.463,E2 -13998.463} C_VEL
LIN {X 0,Y 341.035,Z 264.846,A -85,B 0,C 180,E1 -13998.793,E2 -13998.793} C_VEL
LIN {X 0,Y 340.825,Z 262.078,A -85,B 0,C 180,E1 -14001.787,E2 -14001.787} C_VEL
LIN {X 0,Y 340.699,Z 261.049,A -85,B 0,C 180,E1 -14003.56,E2 -14003.56} C_VEL
LIN {X 0,Y 340.681,Z 261.054,A -85,B 0,C 180,E1 -14006.154,E2 -14006.154} C_VEL
LIN {X 0,Y 340.764,Z 261.042,A -85,B 0,C 180,E1 -14010.333,E2 -14010.333} C_VEL
LIN {X 0,Y 340.794,Z 261.034,A -85,B 0,C 180,E1 -14013.021,E2 -14013.021} C_VEL
LIN {X 0,Y 340.729,Z 261.04,A -85,B 0,C 180,E1 -14016.929,E2 -14016.929} C_VEL
LIN {X 0,Y 340.793,Z 261.036,A -85,B 0,C 180,E1 -14020.735,E2 -14020.735} C_VEL
LIN {X 0,Y 340.778,Z 261.035,A -85,B 0,C 180,E1 -14023.22,E2 -14023.22} C_VEL
LIN {X 0,Y 340.834,Z 261.031,A -85,B 0,C 180,E1 -14026.892,E2 -14026.892} C_VEL
LIN {X 0,Y 340.905,Z 261.021,A -85,B 0,C 180,E1 -14030.509,E2 -14030.509} C_VEL
LIN {X 0,Y 341.05,Z 261.005,A -85,B 0,C 180,E1 -14032.899,E2 -14032.899} C_VEL
LIN {X 0,Y 341.162,Z 260.989,A -85,B 0,C 180,E1 -14037.64,E2 -14037.64} C_VEL
LIN {X 0,Y 341.266,Z 260.974,A -85,B 0,C 180,E1 -14040.001,E2 -14040.001} C_VEL
LIN {X 0,Y 341.162,Z 260.99,A -85,B 0,C 180,E1 -14042.363,E2 -14042.363} C_VEL
LIN {X 0,Y 341.067,Z 261,A -85,B 0,C 180,E1 -14047.103,E2 -14047.103} C_VEL
LIN {X 0,Y 340.864,Z 261.027,A -85,B 0,C 180,E1 -14050.695,E2 -14050.695} C_VEL
LIN {X 0,Y 340.858,Z 261.03,A -85,B 0,C 180,E1 -14054.326,E2 -14054.326} C_VEL
LIN {X 0,Y 340.833,Z 261.035,A -85,B 0,C 180,E1 -14058.468,E2 -14058.468} C_VEL
LIN {X 0,Y 340.75,Z 261.046,A -85,B 0,C 180,E1 -14061.858,E2 -14061.858} C_VEL
LIN {X 0,Y 340.746,Z 261.046,A -85,B 0,C 180,E1 -14065.668,E2 -14065.668} C_VEL
LIN {X 0,Y 340.725,Z 261.047,A -85,B 0,C 180,E1 -14069.674,E2 -14069.674} C_VEL
LIN {X 0,Y 340.69,Z 261.049,A -85,B 0,C 180,E1 -14073.848,E2 -14073.848} C_VEL
LIN {X 0,Y 340.703,Z 261.047,A -85,B 0,C 180,E1 -14076.743,E2 -14076.743} C_VEL
LIN {X 0,Y 340.686,Z 261.043,A -85,B 0,C 180,E1 -14080.248,E2 -14080.248} C_VEL
LIN {X 0,Y 340.684,Z 261.156,A -85,B 0,C 180,E1 -14083.134,E2 -14083.134} C_VEL
LIN {X 0,Y 341.27,Z 264.444,A -85,B 0,C 180,E1 -14086.12,E2 -14086.12} C_VEL
LIN {X 0,Y 341.958,Z 268.456,A -85,B 0,C 180,E1 -14089.504,E2 -14089.504} C_VEL
LIN {X 0,Y 342.589,Z 273.124,A -85,B 0,C 180,E1 -14093.138,E2 -14093.138} C_VEL
LIN {X 0,Y 342.494,Z 275.928,A -85,B 0,C 180,E1 -14095.167,E2 -14095.167} C_VEL
LIN {X 0,Y 341.81,Z 281.669,A -85,B 0,C 180,E1 -14099.068,E2 -14099.068} C_VEL
LIN {X 0,Y 340.964,Z 287.79,A -85,B 0,C 180,E1 -14103.034,E2 -14103.034} C_VEL
LIN {X 0,Y 340.386,Z 293.943,A -85,B 0,C 180,E1 -14106.903,E2 -14106.903} C_VEL
LIN {X 0,Y 340.343,Z 294.619,A -85,B 0,C 180,E1 -14107.319,E2 -14107.319} C_VEL
LIN {X 0,Y 343.897,Z 308.143,A -85,B 0,C 180,E1 -14108.151,E2 -14108.151} C_VEL
LIN {X 0,Y 346.438,Z 320.598,A -85,B 0,C 180,E1 -14109.095,E2 -14109.095} C_VEL
LIN {X 0,Y 347.725,Z 331.557,A -85,B 0,C 180,E1 -14110.059,E2 -14110.059} C_VEL
LIN {X 0,Y 347.846,Z 336.446,A -85,B 0,C 180,E1 -14110.527,E2 -14110.527} C_VEL
LIN {X 0,Y 346.394,Z 347.622,A -85,B 0,C 180,E1 -14111.671,E2 -14111.671} C_VEL
LIN {X 0,Y 344.788,Z 357.735,A -85,B 0,C 180,E1 -14112.962,E2 -14112.962} C_VEL
LIN {X 0,Y 343.411,Z 367.655,A -85,B 0,C 180,E1 -14114.571,E2 -14114.571} C_VEL
LIN {X 0,Y 342.1,Z 376.419,A -85,B 0,C 180,E1 -14116.335,E2 -14116.335} C_VEL
LIN {X 0,Y 340.889,Z 383.471,A -85,B 0,C 180,E1 -14118.103,E2 -14118.103} C_VEL
LIN {X 0,Y 340.129,Z 389.122,A -85,B 0,C 180,E1 -14119.885,E2 -14119.885} C_VEL
LIN {X 0,Y 339.598,Z 393.595,A -85,B 0,C 180,E1 -14121.671,E2 -14121.671} C_VEL
LIN {X 0,Y 339.327,Z 395.962,A -85,B 0,C 180,E1 -14122.862,E2 -14122.862} C_VEL
LIN {X 0,Y 339.154,Z 397.956,A -85,B 0,C 180,E1 -14124.085,E2 -14124.085} C_VEL
LIN {X 0,Y 339.071,Z 399.44,A -85,B 0,C 180,E1 -14125.244,E2 -14125.244} C_VEL
LIN {X 0,Y 339.067,Z 400.527,A -85,B 0,C 180,E1 -14126.435,E2 -14126.435} C_VEL
LIN {X 0,Y 339.008,Z 401.53,A -85,B 0,C 180,E1 -14128.812,E2 -14128.812} C_VEL
LIN {X 0,Y 339.069,Z 401.455,A -85,B 0,C 180,E1 -14130,E2 -14130} C_VEL
LIN {X 0,Y 339.026,Z 400.947,A -85,B 0,C 180,E1 -14131.188,E2 -14131.188} C_VEL
LIN {X 0,Y 339.075,Z 398.727,A -85,B 0,C 180,E1 -14133.565,E2 -14133.565} C_VEL
LIN {X 0,Y 339.089,Z 395.829,A -85,B 0,C 180,E1 -14135.412,E2 -14135.412} C_VEL
LIN {X 0,Y 339.272,Z 392.112,A -85,B 0,C 180,E1 -14137.14,E2 -14137.14} C_VEL
LIN {X 0,Y 339.594,Z 387.145,A -85,B 0,C 180,E1 -14138.929,E2 -14138.929} C_VEL
LIN {X 0,Y 340.116,Z 380.883,A -85,B 0,C 180,E1 -14140.718,E2 -14140.718} C_VEL
LIN {X 0,Y 340.872,Z 373.049,A -85,B 0,C 180,E1 -14142.502,E2 -14142.502} C_VEL
LIN {X 0,Y 341.698,Z 365.031,A -85,B 0,C 180,E1 -14143.985,E2 -14143.985} C_VEL
LIN {X 0,Y 342.643,Z 355.231,A -85,B 0,C 180,E1 -14145.464,E2 -14145.464} C_VEL
LIN {X 0,Y 343.635,Z 344.323,A -85,B 0,C 180,E1 -14146.791,E2 -14146.791} C_VEL
LIN {X 0,Y 344.853,Z 332.112,A -85,B 0,C 180,E1 -14147.935,E2 -14147.935} C_VEL
LIN {X 0,Y 343.399,Z 319.082,A -85,B 0,C 180,E1 -14148.968,E2 -14148.968} C_VEL
LIN {X 0,Y 341.569,Z 306.015,A -85,B 0,C 180,E1 -14149.744,E2 -14149.744} C_VEL
LIN {X 0,Y 339.725,Z 295.045,A -85,B 0,C 180,E1 -14150.234,E2 -14150.234} C_VEL
LIN {X 0,Y 340.051,Z 290.137,A -85,B 0,C 180,E1 -14153.121,E2 -14153.121} C_VEL
LIN {X 0,Y 340.578,Z 283.633,A -85,B 0,C 180,E1 -14156.999,E2 -14156.999} C_VEL
LIN {X 0,Y 341.202,Z 277.079,A -85,B 0,C 180,E1 -14160.993,E2 -14160.993} C_VEL
LIN {X 0,Y 341.822,Z 271.244,A -85,B 0,C 180,E1 -14164.671,E2 -14164.671} C_VEL
LIN {X 0,Y 341.778,Z 267.201,A -85,B 0,C 180,E1 -14167.343,E2 -14167.343} C_VEL
LIN {X 0,Y 341.104,Z 262.922,A -85,B 0,C 180,E1 -14170.328,E2 -14170.328} C_VEL
LIN {X 0,Y 340.74,Z 261.043,A -85,B 0,C 180,E1 -14171.801,E2 -14171.801} C_VEL
LIN {X 0,Y 340.628,Z 261.053,A -85,B 0,C 180,E1 -14175.451,E2 -14175.451} C_VEL
LIN {X 0,Y 340.643,Z 261.054,A -85,B 0,C 180,E1 -14178.683,E2 -14178.683} C_VEL
LIN {X 0,Y 340.716,Z 261.041,A -85,B 0,C 180,E1 -14181.769,E2 -14181.769} C_VEL
LIN {X 0,Y 340.719,Z 261.04,A -85,B 0,C 180,E1 -14185.594,E2 -14185.594} C_VEL
LIN {X 0,Y 340.69,Z 261.047,A -85,B 0,C 180,E1 -14188.953,E2 -14188.953} C_VEL
LIN {X 0,Y 340.715,Z 261.042,A -85,B 0,C 180,E1 -14193.011,E2 -14193.011} C_VEL
LIN {X 0,Y 340.736,Z 261.038,A -85,B 0,C 180,E1 -14195.636,E2 -14195.636} C_VEL
LIN {X 0,Y 340.728,Z 261.039,A -85,B 0,C 180,E1 -14199.472,E2 -14199.472} C_VEL
LIN {X 0,Y 340.853,Z 261.026,A -85,B 0,C 180,E1 -14201.983,E2 -14201.983} C_VEL
LIN {X 0,Y 340.865,Z 261.024,A -85,B 0,C 180,E1 -14205.704,E2 -14205.704} C_VEL
LIN {X 0,Y 340.865,Z 261.022,A -85,B 0,C 180,E1 -14209.305,E2 -14209.305} C_VEL
LIN {X 0,Y 341.053,Z 260.999,A -85,B 0,C 180,E1 -14212.896,E2 -14212.896} C_VEL
LIN {X 0,Y 341.162,Z 260.988,A -85,B 0,C 180,E1 -14217.637,E2 -14217.637} C_VEL
LIN {X 0,Y 341.31,Z 260.972,A -85,B 0,C 180,E1 -14219.999,E2 -14219.999} C_VEL
LIN {X 0,Y 341.162,Z 260.986,A -85,B 0,C 180,E1 -14222.36,E2 -14222.36} C_VEL
LIN {X 0,Y 341.067,Z 260.998,A -85,B 0,C 180,E1 -14227.1,E2 -14227.1} C_VEL
LIN {X 0,Y 340.862,Z 261.022,A -85,B 0,C 180,E1 -14230.693,E2 -14230.693} C_VEL
LIN {X 0,Y 340.854,Z 261.024,A -85,B 0,C 180,E1 -14234.324,E2 -14234.324} C_VEL
LIN {X 0,Y 340.827,Z 261.027,A -85,B 0,C 180,E1 -14238.465,E2 -14238.465} C_VEL
LIN {X 0,Y 340.744,Z 261.039,A -85,B 0,C 180,E1 -14241.856,E2 -14241.856} C_VEL
LIN {X 0,Y 340.762,Z 261.037,A -85,B 0,C 180,E1 -14245.663,E2 -14245.663} C_VEL
LIN {X 0,Y 340.732,Z 261.039,A -85,B 0,C 180,E1 -14248.319,E2 -14248.319} C_VEL
LIN {X 0,Y 340.693,Z 261.048,A -85,B 0,C 180,E1 -14251.043,E2 -14251.043} C_VEL
LIN {X 0,Y 340.707,Z 261.046,A -85,B 0,C 180,E1 -14255.278,E2 -14255.278} C_VEL
LIN {X 0,Y 340.707,Z 261.043,A -85,B 0,C 180,E1 -14258.387,E2 -14258.387} C_VEL
LIN {X 0,Y 340.714,Z 261.043,A -85,B 0,C 180,E1 -14261.303,E2 -14261.303} C_VEL
LIN {X 0,Y 340.709,Z 261.044,A -85,B 0,C 180,E1 -14264.532,E2 -14264.532} C_VEL
LIN {X 0,Y 340.675,Z 261.051,A -85,B 0,C 180,E1 -14268.69,E2 -14268.69} C_VEL
LIN {X 0,Y 340.724,Z 261.04,A -85,B 0,C 180,E1 -14271.772,E2 -14271.772} C_VEL
LIN {X 0,Y 340.711,Z 261.041,A -85,B 0,C 180,E1 -14275.595,E2 -14275.595} C_VEL
LIN {X 0,Y 340.686,Z 261.046,A -85,B 0,C 180,E1 -14278.955,E2 -14278.955} C_VEL
LIN {X 0,Y 340.748,Z 261.042,A -85,B 0,C 180,E1 -14282.48,E2 -14282.48} C_VEL
LIN {X 0,Y 340.68,Z 261.046,A -85,B 0,C 180,E1 -14285.633,E2 -14285.633} C_VEL
LIN {X 0,Y 340.511,Z 261.108,A -85,B 0,C 180,E1 -14288.24,E2 -14288.24} C_VEL
LIN {X 0,Y 340.362,Z 265.238,A -85,B 0,C 180,E1 -14291.957,E2 -14291.957} C_VEL
LIN {X 0,Y 340.143,Z 270.091,A -85,B 0,C 180,E1 -14296.186,E2 -14296.186} C_VEL
LIN {X 0,Y 339.882,Z 275.158,A -85,B 0,C 180,E1 -14300.478,E2 -14300.478} C_VEL
LIN {X 0,Y 339.914,Z 278.038,A -85,B 0,C 180,E1 -14302.874,E2 -14302.874} C_VEL
LIN {X 0,Y 342.845,Z 292.152,A -85,B 0,C 180,E1 -14303.594,E2 -14303.594} C_VEL
LIN {X 0,Y 344.853,Z 304.727,A -85,B 0,C 180,E1 -14304.445,E2 -14304.445} C_VEL
LIN {X 0,Y 345.518,Z 310.305,A -85,B 0,C 180,E1 -14304.895,E2 -14304.895} C_VEL
LIN {X 0,Y 344.58,Z 321.775,A -85,B 0,C 180,E1 -14305.906,E2 -14305.906} C_VEL
LIN {X 0,Y 343.459,Z 333.373,A -85,B 0,C 180,E1 -14307.214,E2 -14307.214} C_VEL
LIN {X 0,Y 342.519,Z 342.722,A -85,B 0,C 180,E1 -14308.53,E2 -14308.53} C_VEL
LIN {X 0,Y 341.645,Z 351.252,A -85,B 0,C 180,E1 -14310,E2 -14310} C_VEL
LIN {X 0,Y 340.688,Z 359.563,A -85,B 0,C 180,E1 -14311.773,E2 -14311.773} C_VEL
LIN {X 0,Y 340.106,Z 366.246,A -85,B 0,C 180,E1 -14313.554,E2 -14313.554} C_VEL
LIN {X 0,Y 339.681,Z 371.589,A -85,B 0,C 180,E1 -14315.342,E2 -14315.342} C_VEL
LIN {X 0,Y 339.37,Z 375.765,A -85,B 0,C 180,E1 -14317.137,E2 -14317.137} C_VEL
LIN {X 0,Y 339.169,Z 377.978,A -85,B 0,C 180,E1 -14318.34,E2 -14318.34} C_VEL
LIN {X 0,Y 339.003,Z 379.704,A -85,B 0,C 180,E1 -14319.546,E2 -14319.546} C_VEL
LIN {X 0,Y 338.938,Z 381.019,A -85,B 0,C 180,E1 -14320.755,E2 -14320.755} C_VEL
LIN {X 0,Y 338.943,Z 382.366,A -85,B 0,C 180,E1 -14322.964,E2 -14322.964} C_VEL
LIN {X 0,Y 338.92,Z 382.474,A -85,B 0,C 180,E1 -14324.408,E2 -14324.408} C_VEL
LIN {X 0,Y 338.95,Z 382.137,A -85,B 0,C 180,E1 -14325.637,E2 -14325.637} C_VEL
LIN {X 0,Y 339.233,Z 380.675,A -85,B 0,C 180,E1 -14327.643,E2 -14327.643} C_VEL
LIN {X 0,Y 339.7,Z 377.532,A -85,B 0,C 180,E1 -14329.96,E2 -14329.96} C_VEL
LIN {X 0,Y 340.28,Z 373.8,A -85,B 0,C 180,E1 -14331.824,E2 -14331.824} C_VEL
LIN {X 0,Y 341.056,Z 368.857,A -85,B 0,C 180,E1 -14333.692,E2 -14333.692} C_VEL
LIN {X 0,Y 342.077,Z 362.541,A -85,B 0,C 180,E1 -14335.559,E2 -14335.559} C_VEL
LIN {X 0,Y 343.383,Z 354.581,A -85,B 0,C 180,E1 -14337.419,E2 -14337.419} C_VEL
LIN {X 0,Y 344.817,Z 345.562,A -85,B 0,C 180,E1 -14339.088,E2 -14339.088} C_VEL
LIN {X 0,Y 346.232,Z 336.162,A -85,B 0,C 180,E1 -14340.494,E2 -14340.494} C_VEL
LIN {X 0,Y 347.675,Z 325.485,A -85,B 0,C 180,E1 -14341.781,E2 -14341.781} C_VEL
LIN {X 0,Y 349.066,Z 313.224,A -85,B 0,C 180,E1 -14342.929,E2 -14342.929} C_VEL
LIN {X 0,Y 347.179,Z 302.777,A -85,B 0,C 180,E1 -14343.908,E2 -14343.908} C_VEL
LIN {X 0,Y 343.752,Z 289.943,A -85,B 0,C 180,E1 -14344.956,E2 -14344.956} C_VEL
LIN {X 0,Y 340.054,Z 278.884,A -85,B 0,C 180,E1 -14345.72,E2 -14345.72} C_VEL
LIN {X 0,Y 339.99,Z 278.509,A -85,B 0,C 180,E1 -14345.739,E2 -14345.739} C_VEL
LIN {X 0,Y 340.345,Z 274.035,A -85,B 0,C 180,E1 -14349.801,E2 -14349.801} C_VEL
LIN {X 0,Y 340.689,Z 269.841,A -85,B 0,C 180,E1 -14353.782,E2 -14353.782} C_VEL
LIN {X 0,Y 340.931,Z 267.392,A -85,B 0,C 180,E1 -14356.177,E2 -14356.177} C_VEL
LIN {X 0,Y 341.035,Z 264.846,A -85,B 0,C 180,E1 -14358.793,E2 -14358.793} C_VEL
LIN {X 0,Y 340.313,Z 264.055,A -85,B 0,C 180,E1 -14359.768,E2 -14359.768} C_VEL
LIN {X 0,Y 337.353,Z 263.057,A -85,B 0,C 180,E1 -14361.356,E2 -14361.356} C_VEL
LIN {X 0,Y 334.849,Z 262.333,A -85,B 0,C 180,E1 -14362.647,E2 -14362.647} C_VEL
LIN {X 0,Y 333.757,Z 261.958,A -85,B 0,C 180,E1 -14363.651,E2 -14363.651} C_VEL
LIN {X 0,Y 333.658,Z 261.925,A -85,B 0,C 180,E1 -14363.991,E2 -14363.991} C_VEL
LIN {X 0,Y 333.632,Z 261.932,A -85,B 0,C 180,E1 -14367.414,E2 -14367.414} C_VEL
LIN {X 0,Y 333.7,Z 261.918,A -85,B 0,C 180,E1 -14371.029,E2 -14371.029} C_VEL
LIN {X 0,Y 333.726,Z 261.916,A -85,B 0,C 180,E1 -14373.755,E2 -14373.755} C_VEL
LIN {X 0,Y 333.712,Z 261.918,A -85,B 0,C 180,E1 -14377.914,E2 -14377.914} C_VEL
LIN {X 0,Y 333.785,Z 261.907,A -85,B 0,C 180,E1 -14381.591,E2 -14381.591} C_VEL
LIN {X 0,Y 333.799,Z 261.902,A -85,B 0,C 180,E1 -14385.578,E2 -14385.578} C_VEL
LIN {X 0,Y 333.824,Z 261.903,A -85,B 0,C 180,E1 -14389.079,E2 -14389.079} C_VEL
LIN {X 0,Y 333.997,Z 261.883,A -85,B 0,C 180,E1 -14392.748,E2 -14392.748} C_VEL
LIN {X 0,Y 333.802,Z 261.905,A -85,B 0,C 180,E1 -14395.17,E2 -14395.17} C_VEL
LIN {X 0,Y 334.099,Z 261.869,A -85,B 0,C 180,E1 -14397.59,E2 -14397.59} C_VEL
LIN {X 0,Y 334.218,Z 261.852,A -85,B 0,C 180,E1 -14400.001,E2 -14400.001} C_VEL
LIN {X 0,Y 334.099,Z 261.869,A -85,B 0,C 180,E1 -14402.413,E2 -14402.413} C_VEL
LIN {X 0,Y 334.017,Z 261.878,A -85,B 0,C 180,E1 -14407.254,E2 -14407.254} C_VEL
LIN {X 0,Y 333.827,Z 261.905,A -85,B 0,C 180,E1 -14410.924,E2 -14410.924} C_VEL
LIN {X 0,Y 333.803,Z 261.907,A -85,B 0,C 180,E1 -14414.636,E2 -14414.636} C_VEL
LIN {X 0,Y 333.792,Z 261.911,A -85,B 0,C 180,E1 -14418.657,E2 -14418.657} C_VEL
LIN {X 0,Y 333.688,Z 261.924,A -85,B 0,C 180,E1 -14422.28,E2 -14422.28} C_VEL
LIN {X 0,Y 333.706,Z 261.924,A -85,B 0,C 180,E1 -14425.099,E2 -14425.099} C_VEL
LIN {X 0,Y 333.667,Z 261.928,A -85,B 0,C 180,E1 -14428.978,E2 -14428.978} C_VEL
LIN {X 0,Y 333.641,Z 261.928,A -85,B 0,C 180,E1 -14432.588,E2 -14432.588} C_VEL
LIN {X 0,Y 333.674,Z 261.922,A -85,B 0,C 180,E1 -14436.141,E2 -14436.141} C_VEL
LIN {X 0,Y 333.645,Z 261.925,A -85,B 0,C 180,E1 -14439.194,E2 -14439.194} C_VEL
LIN {X 0,Y 333.637,Z 261.963,A -85,B 0,C 180,E1 -14442.502,E2 -14442.502} C_VEL
LIN {X 0,Y 334.314,Z 265.792,A -85,B 0,C 180,E1 -14446.075,E2 -14446.075} C_VEL
LIN {X 0,Y 334.974,Z 269.682,A -85,B 0,C 180,E1 -14449.429,E2 -14449.429} C_VEL
LIN {X 0,Y 335.53,Z 273.834,A -85,B 0,C 180,E1 -14452.746,E2 -14452.746} C_VEL
LIN {X 0,Y 335.398,Z 277.633,A -85,B 0,C 180,E1 -14455.546,E2 -14455.546} C_VEL
LIN {X 0,Y 334.681,Z 283.251,A -85,B 0,C 180,E1 -14459.427,E2 -14459.427} C_VEL
LIN {X 0,Y 333.917,Z 288.782,A -85,B 0,C 180,E1 -14463.096,E2 -14463.096} C_VEL
LIN {X 0,Y 333.348,Z 294.409,A -85,B 0,C 180,E1 -14466.709,E2 -14466.709} C_VEL
LIN {X 0,Y 337.111,Z 308.251,A -85,B 0,C 180,E1 -14467.609,E2 -14467.609} C_VEL
LIN {X 0,Y 339.662,Z 320.983,A -85,B 0,C 180,E1 -14468.61,E2 -14468.61} C_VEL
LIN {X 0,Y 340.888,Z 330.595,A -85,B 0,C 180,E1 -14469.484,E2 -14469.484} C_VEL
LIN {X 0,Y 341.196,Z 337.088,A -85,B 0,C 180,E1 -14470.132,E2 -14470.132} C_VEL
LIN {X 0,Y 339.687,Z 348.108,A -85,B 0,C 180,E1 -14471.296,E2 -14471.296} C_VEL
LIN {X 0,Y 338.184,Z 357.063,A -85,B 0,C 180,E1 -14472.463,E2 -14472.463} C_VEL
LIN {X 0,Y 336.832,Z 366.039,A -85,B 0,C 180,E1 -14473.907,E2 -14473.907} C_VEL
LIN {X 0,Y 335.41,Z 375.231,A -85,B 0,C 180,E1 -14475.747,E2 -14475.747} C_VEL
LIN {X 0,Y 334.129,Z 382.477,A -85,B 0,C 180,E1 -14477.55,E2 -14477.55} C_VEL
LIN {X 0,Y 333.13,Z 389.134,A -85,B 0,C 180,E1 -14479.67,E2 -14479.67} C_VEL
LIN {X 0,Y 332.564,Z 393.555,A -85,B 0,C 180,E1 -14481.493,E2 -14481.493} C_VEL
LIN {X 0,Y 332.268,Z 395.898,A -85,B 0,C 180,E1 -14482.709,E2 -14482.709} C_VEL
LIN {X 0,Y 332.066,Z 398.102,A -85,B 0,C 180,E1 -14484.124,E2 -14484.124} C_VEL
LIN {X 0,Y 331.971,Z 400.376,A -85,B 0,C 180,E1 -14486.359,E2 -14486.359} C_VEL
LIN {X 0,Y 331.914,Z 401.339,A -85,B 0,C 180,E1 -14488.787,E2 -14488.787} C_VEL
LIN {X 0,Y 331.972,Z 401.236,A -85,B 0,C 180,E1 -14490,E2 -14490} C_VEL
LIN {X 0,Y 331.932,Z 400.697,A -85,B 0,C 180,E1 -14491.213,E2 -14491.213} C_VEL
LIN {X 0,Y 332.001,Z 398.436,A -85,B 0,C 180,E1 -14493.641,E2 -14493.641} C_VEL
LIN {X 0,Y 332.085,Z 394.774,A -85,B 0,C 180,E1 -14495.908,E2 -14495.908} C_VEL
LIN {X 0,Y 332.312,Z 390.191,A -85,B 0,C 180,E1 -14497.901,E2 -14497.901} C_VEL
LIN {X 0,Y 332.833,Z 383.735,A -85,B 0,C 180,E1 -14500.032,E2 -14500.032} C_VEL
LIN {X 0,Y 333.426,Z 376.657,A -85,B 0,C 180,E1 -14501.859,E2 -14501.859} C_VEL
LIN {X 0,Y 334.425,Z 367.794,A -85,B 0,C 180,E1 -14503.675,E2 -14503.675} C_VEL
LIN {X 0,Y 335.355,Z 358.216,A -85,B 0,C 180,E1 -14505.261,E2 -14505.261} C_VEL
LIN {X 0,Y 336.291,Z 348.65,A -85,B 0,C 180,E1 -14506.543,E2 -14506.543} C_VEL
LIN {X 0,Y 337.44,Z 337.492,A -85,B 0,C 180,E1 -14507.734,E2 -14507.734} C_VEL
LIN {X 0,Y 337.881,Z 332.539,A -85,B 0,C 180,E1 -14508.18,E2 -14508.18} C_VEL
LIN {X 0,Y 336.674,Z 321.338,A -85,B 0,C 180,E1 -14509.11,E2 -14509.11} C_VEL
LIN {X 0,Y 334.873,Z 307.861,A -85,B 0,C 180,E1 -14509.981,E2 -14509.981} C_VEL
LIN {X 0,Y 332.705,Z 294.856,A -85,B 0,C 180,E1 -14510.599,E2 -14510.599} C_VEL
LIN {X 0,Y 333.121,Z 288.763,A -85,B 0,C 180,E1 -14514.269,E2 -14514.269} C_VEL
LIN {X 0,Y 333.59,Z 283.04,A -85,B 0,C 180,E1 -14517.765,E2 -14517.765} C_VEL
LIN {X 0,Y 334.273,Z 276.761,A -85,B 0,C 180,E1 -14521.709,E2 -14521.709} C_VEL
LIN {X 0,Y 334.804,Z 271.592,A -85,B 0,C 180,E1 -14525.047,E2 -14525.047} C_VEL
LIN {X 0,Y 334.733,Z 267.973,A -85,B 0,C 180,E1 -14527.508,E2 -14527.508} C_VEL
LIN {X 0,Y 333.971,Z 263.453,A -85,B 0,C 180,E1 -14530.748,E2 -14530.748} C_VEL
LIN {X 0,Y 333.689,Z 261.922,A -85,B 0,C 180,E1 -14531.966,E2 -14531.966} C_VEL
LIN {X 0,Y 333.585,Z 261.929,A -85,B 0,C 180,E1 -14535.952,E2 -14535.952} C_VEL
LIN {X 0,Y 333.596,Z 261.93,A -85,B 0,C 180,E1 -14539.324,E2 -14539.324} C_VEL
LIN {X 0,Y 333.659,Z 261.922,A -85,B 0,C 180,E1 -14543.168,E2 -14543.168} C_VEL
LIN {X 0,Y 333.67,Z 261.919,A -85,B 0,C 180,E1 -14545.339,E2 -14545.339} C_VEL
LIN {X 0,Y 333.627,Z 261.926,A -85,B 0,C 180,E1 -14548.22,E2 -14548.22} C_VEL
LIN {X 0,Y 333.65,Z 261.923,A -85,B 0,C 180,E1 -14551.021,E2 -14551.021} C_VEL
LIN {X 0,Y 333.692,Z 261.916,A -85,B 0,C 180,E1 -14555.087,E2 -14555.087} C_VEL
LIN {X 0,Y 333.661,Z 261.92,A -85,B 0,C 180,E1 -14559.017,E2 -14559.017} C_VEL
LIN {X 0,Y 333.789,Z 261.904,A -85,B 0,C 180,E1 -14561.588,E2 -14561.588} C_VEL
LIN {X 0,Y 333.804,Z 261.903,A -85,B 0,C 180,E1 -14565.575,E2 -14565.575} C_VEL
LIN {X 0,Y 333.828,Z 261.899,A -85,B 0,C 180,E1 -14569.076,E2 -14569.076} C_VEL
LIN {X 0,Y 334,Z 261.878,A -85,B 0,C 180,E1 -14572.746,E2 -14572.746} C_VEL
LIN {X 0,Y 333.801,Z 261.902,A -85,B 0,C 180,E1 -14575.168,E2 -14575.168} C_VEL
LIN {X 0,Y 334.099,Z 261.867,A -85,B 0,C 180,E1 -14577.587,E2 -14577.587} C_VEL
LIN {X 0,Y 334.26,Z 261.849,A -85,B 0,C 180,E1 -14579.999,E2 -14579.999} C_VEL
LIN {X 0,Y 334.1,Z 261.866,A -85,B 0,C 180,E1 -14582.41,E2 -14582.41} C_VEL
LIN {X 0,Y 334.017,Z 261.877,A -85,B 0,C 180,E1 -14587.251,E2 -14587.251} C_VEL
LIN {X 0,Y 333.825,Z 261.899,A -85,B 0,C 180,E1 -14590.921,E2 -14590.921} C_VEL
LIN {X 0,Y 333.799,Z 261.902,A -85,B 0,C 180,E1 -14594.633,E2 -14594.633} C_VEL
LIN {X 0,Y 333.786,Z 261.904,A -85,B 0,C 180,E1 -14598.653,E2 -14598.653} C_VEL
LIN {X 0,Y 333.683,Z 261.917,A -85,B 0,C 180,E1 -14602.277,E2 -14602.277} C_VEL
LIN {X 0,Y 333.726,Z 261.911,A -85,B 0,C 180,E1 -14606.245,E2 -14606.245} C_VEL
LIN {X 0,Y 333.701,Z 261.918,A -85,B 0,C 180,E1 -14608.971,E2 -14608.971} C_VEL
LIN {X 0,Y 333.633,Z 261.924,A -85,B 0,C 180,E1 -14612.586,E2 -14612.586} C_VEL
LIN {X 0,Y 333.665,Z 261.919,A -85,B 0,C 180,E1 -14616.138,E2 -14616.138} C_VEL
LIN {X 0,Y 333.673,Z 261.922,A -85,B 0,C 180,E1 -14619.186,E2 -14619.186} C_VEL
LIN {X 0,Y 333.677,Z 261.92,A -85,B 0,C 180,E1 -14622.51,E2 -14622.51} C_VEL
LIN {X 0,Y 333.623,Z 261.924,A -85,B 0,C 180,E1 -14625.961,E2 -14625.961} C_VEL
LIN {X 0,Y 333.636,Z 261.924,A -85,B 0,C 180,E1 -14629.315,E2 -14629.315} C_VEL
LIN {X 0,Y 333.655,Z 261.922,A -85,B 0,C 180,E1 -14633.167,E2 -14633.167} C_VEL
LIN {X 0,Y 333.625,Z 261.928,A -85,B 0,C 180,E1 -14636.791,E2 -14636.791} C_VEL
LIN {X 0,Y 333.683,Z 261.917,A -85,B 0,C 180,E1 -14639.712,E2 -14639.712} C_VEL
LIN {X 0,Y 333.713,Z 261.919,A -85,B 0,C 180,E1 -14642.399,E2 -14642.399} C_VEL
LIN {X 0,Y 333.653,Z 261.921,A -85,B 0,C 180,E1 -14645.085,E2 -14645.085} C_VEL
LIN {X 0,Y 333.476,Z 262.112,A -85,B 0,C 180,E1 -14648.328,E2 -14648.328} C_VEL
LIN {X 0,Y 333.356,Z 265.627,A -85,B 0,C 180,E1 -14651.565,E2 -14651.565} C_VEL
LIN {X 0,Y 333.092,Z 270.683,A -85,B 0,C 180,E1 -14656.056,E2 -14656.056} C_VEL
LIN {X 0,Y 332.825,Z 275.595,A -85,B 0,C 180,E1 -14660.275,E2 -14660.275} C_VEL
LIN {X 0,Y 332.845,Z 278.355,A -85,B 0,C 180,E1 -14662.527,E2 -14662.527} C_VEL
LIN {X 0,Y 335.584,Z 291.303,A -85,B 0,C 180,E1 -14663.192,E2 -14663.192} C_VEL
LIN {X 0,Y 337.683,Z 303.529,A -85,B 0,C 180,E1 -14664.027,E2 -14664.027} C_VEL
LIN {X 0,Y 338.605,Z 311.051,A -85,B 0,C 180,E1 -14664.641,E2 -14664.641} C_VEL
LIN {X 0,Y 337.642,Z 322.396,A -85,B 0,C 180,E1 -14665.673,E2 -14665.673} C_VEL
LIN {X 0,Y 336.499,Z 333.922,A -85,B 0,C 180,E1 -14667.007,E2 -14667.007} C_VEL
LIN {X 0,Y 335.664,Z 342.235,A -85,B 0,C 180,E1 -14668.2,E2 -14668.2} C_VEL
LIN {X 0,Y 334.703,Z 350.908,A -85,B 0,C 180,E1 -14669.699,E2 -14669.699} C_VEL
LIN {X 0,Y 333.697,Z 359.339,A -85,B 0,C 180,E1 -14671.508,E2 -14671.508} C_VEL
LIN {X 0,Y 333.084,Z 366.1,A -85,B 0,C 180,E1 -14673.326,E2 -14673.326} C_VEL
LIN {X 0,Y 332.567,Z 372.322,A -85,B 0,C 180,E1 -14675.457,E2 -14675.457} C_VEL
LIN {X 0,Y 332.25,Z 376.377,A -85,B 0,C 180,E1 -14677.291,E2 -14677.291} C_VEL
LIN {X 0,Y 332.039,Z 378.48,A -85,B 0,C 180,E1 -14678.52,E2 -14678.52} C_VEL
LIN {X 0,Y 331.884,Z 380.149,A -85,B 0,C 180,E1 -14679.753,E2 -14679.753} C_VEL
LIN {X 0,Y 331.832,Z 381.409,A -85,B 0,C 180,E1 -14680.988,E2 -14680.988} C_VEL
LIN {X 0,Y 331.862,Z 382.574,A -85,B 0,C 180,E1 -14683.062,E2 -14683.062} C_VEL
LIN {X 0,Y 331.83,Z 382.651,A -85,B 0,C 180,E1 -14684.723,E2 -14684.723} C_VEL
LIN {X 0,Y 331.893,Z 382.259,A -85,B 0,C 180,E1 -14685.978,E2 -14685.978} C_VEL
LIN {X 0,Y 332.173,Z 380.885,A -85,B 0,C 180,E1 -14687.813,E2 -14687.813} C_VEL
LIN {X 0,Y 332.733,Z 377.377,A -85,B 0,C 180,E1 -14690.396,E2 -14690.396} C_VEL
LIN {X 0,Y 333.389,Z 373.524,A -85,B 0,C 180,E1 -14692.299,E2 -14692.299} C_VEL
LIN {X 0,Y 334.24,Z 368.448,A -85,B 0,C 180,E1 -14694.206,E2 -14694.206} C_VEL
LIN {X 0,Y 335.419,Z 361.991,A -85,B 0,C 180,E1 -14696.104,E2 -14696.104} C_VEL
LIN {X 0,Y 336.804,Z 353.779,A -85,B 0,C 180,E1 -14698.001,E2 -14698.001} C_VEL
LIN {X 0,Y 338.274,Z 344.883,A -85,B 0,C 180,E1 -14699.646,E2 -14699.646} C_VEL
LIN {X 0,Y 339.836,Z 334.894,A -85,B 0,C 180,E1 -14701.131,E2 -14701.131} C_VEL
LIN {X 0,Y 341.354,Z 323.897,A -85,B 0,C 180,E1 -14702.424,E2 -14702.424} C_VEL
LIN {X 0,Y 342.464,Z 314.733,A -85,B 0,C 180,E1 -14703.294,E2 -14703.294} C_VEL
LIN {X 0,Y 340.507,Z 303.973,A -85,B 0,C 180,E1 -14704.355,E2 -14704.355} C_VEL
LIN {X 0,Y 337.209,Z 291.497,A -85,B 0,C 180,E1 -14705.425,E2 -14705.425} C_VEL
LIN {X 0,Y 332.987,Z 278.694,A -85,B 0,C 180,E1 -14706.36,E2 -14706.36} C_VEL
LIN {X 0,Y 333.244,Z 275.581,A -85,B 0,C 180,E1 -14709.248,E2 -14709.248} C_VEL
LIN {X 0,Y 333.547,Z 272.21,A -85,B 0,C 180,E1 -14712.487,E2 -14712.487} C_VEL
LIN {X 0,Y 333.923,Z 268.64,A -85,B 0,C 180,E1 -14716.012,E2 -14716.012} C_VEL
LIN {X 0,Y 334.012,Z 265.524,A -85,B 0,C 180,E1 -14719.289,E2 -14719.289} C_VEL
LIN {X 0,Y 333.738,Z 262.775,A -85,B 0,C 180,E1 -14722.363,E2 -14722.363} C_VEL
LIN {X 0,Y 333.664,Z 262.086,A -85,B 0,C 180,E1 -14723.166,E2 -14723.166} C_VEL
LIN {X 0,Y 333.658,Z 261.925,A -85,B 0,C 180,E1 -14723.991,E2 -14723.991} C_VEL
LIN {X 0,Y 332.947,Z 262.016,A -85,B 0,C 180,E1 -14725,E2 -14725} C_VEL
LIN {X 0,Y 330.038,Z 262.38,A -85,B 0,C 180,E1 -14726.639,E2 -14726.639} C_VEL
LIN {X 0,Y 327.637,Z 262.679,A -85,B 0,C 180,E1 -14727.968,E2 -14727.968} C_VEL
LIN {X 0,Y 326.669,Z 262.798,A -85,B 0,C 180,E1 -14728.996,E2 -14728.996} C_VEL
LIN {X 0,Y 326.623,Z 262.802,A -85,B 0,C 180,E1 -14729.344,E2 -14729.344} C_VEL
LIN {X 0,Y 326.675,Z 262.793,A -85,B 0,C 180,E1 -14733.143,E2 -14733.143} C_VEL
LIN {X 0,Y 326.652,Z 262.797,A -85,B 0,C 180,E1 -14735.873,E2 -14735.873} C_VEL
LIN {X 0,Y 326.674,Z 262.791,A -85,B 0,C 180,E1 -14739.868,E2 -14739.868} C_VEL
LIN {X 0,Y 326.69,Z 262.788,A -85,B 0,C 180,E1 -14742.473,E2 -14742.473} C_VEL
LIN {X 0,Y 326.749,Z 262.782,A -85,B 0,C 180,E1 -14746.316,E2 -14746.316} C_VEL
LIN {X 0,Y 326.797,Z 262.779,A -85,B 0,C 180,E1 -14750.095,E2 -14750.095} C_VEL
LIN {X 0,Y 326.98,Z 262.754,A -85,B 0,C 180,E1 -14753.832,E2 -14753.832} C_VEL
LIN {X 0,Y 327.04,Z 262.748,A -85,B 0,C 180,E1 -14757.538,E2 -14757.538} C_VEL
LIN {X 0,Y 327.17,Z 262.73,A -85,B 0,C 180,E1 -14760.001,E2 -14760.001} C_VEL
LIN {X 0,Y 327.04,Z 262.749,A -85,B 0,C 180,E1 -14762.465,E2 -14762.465} C_VEL
LIN {X 0,Y 326.988,Z 262.753,A -85,B 0,C 180,E1 -14766.171,E2 -14766.171} C_VEL
LIN {X 0,Y 326.909,Z 262.764,A -85,B 0,C 180,E1 -14768.657,E2 -14768.657} C_VEL
LIN {X 0,Y 326.729,Z 262.788,A -85,B 0,C 180,E1 -14772.423,E2 -14772.423} C_VEL
LIN {X 0,Y 326.749,Z 262.786,A -85,B 0,C 180,E1 -14774.959,E2 -14774.959} C_VEL
LIN {X 0,Y 326.729,Z 262.79,A -85,B 0,C 180,E1 -14778.84,E2 -14778.84} C_VEL
LIN {X 0,Y 326.617,Z 262.806,A -85,B 0,C 180,E1 -14782.789,E2 -14782.789} C_VEL
LIN {X 0,Y 326.643,Z 262.803,A -85,B 0,C 180,E1 -14785.489,E2 -14785.489} C_VEL
LIN {X 0,Y 326.627,Z 262.804,A -85,B 0,C 180,E1 -14788.255,E2 -14788.255} C_VEL
LIN {X 0,Y 326.571,Z 262.81,A -85,B 0,C 180,E1 -14791.099,E2 -14791.099} C_VEL
LIN {X 0,Y 326.605,Z 262.804,A -85,B 0,C 180,E1 -14794.021,E2 -14794.021} C_VEL
LIN {X 0,Y 326.626,Z 262.8,A -85,B 0,C 180,E1 -14797.24,E2 -14797.24} C_VEL
LIN {X 0,Y 326.577,Z 262.803,A -85,B 0,C 180,E1 -14801.133,E2 -14801.133} C_VEL
LIN {X 0,Y 326.619,Z 262.986,A -85,B 0,C 180,E1 -14802.048,E2 -14802.048} C_VEL
LIN {X 0,Y 327.162,Z 266.189,A -85,B 0,C 180,E1 -14805.147,E2 -14805.147} C_VEL
LIN {X 0,Y 327.85,Z 270.051,A -85,B 0,C 180,E1 -14808.616,E2 -14808.616} C_VEL
LIN {X 0,Y 328.469,Z 274.543,A -85,B 0,C 180,E1 -14812.343,E2 -14812.343} C_VEL
LIN {X 0,Y 328.508,Z 277.641,A -85,B 0,C 180,E1 -14814.717,E2 -14814.717} C_VEL
LIN {X 0,Y 327.986,Z 281.656,A -85,B 0,C 180,E1 -14817.61,E2 -14817.61} C_VEL
LIN {X 0,Y 327.359,Z 285.706,A -85,B 0,C 180,E1 -14820.411,E2 -14820.411} C_VEL
LIN {X 0,Y 326.716,Z 290.79,A -85,B 0,C 180,E1 -14823.835,E2 -14823.835} C_VEL
LIN {X 0,Y 326.413,Z 294.207,A -85,B 0,C 180,E1 -14826.083,E2 -14826.083} C_VEL
LIN {X 0,Y 328.01,Z 300.001,A -85,B 0,C 180,E1 -14826.44,E2 -14826.44} C_VEL
LIN {X 0,Y 331.135,Z 311.97,A -85,B 0,C 180,E1 -14827.312,E2 -14827.312} C_VEL
LIN {X 0,Y 333.313,Z 323.608,A -85,B 0,C 180,E1 -14828.303,E2 -14828.303} C_VEL
LIN {X 0,Y 334.435,Z 334.679,A -85,B 0,C 180,E1 -14829.391,E2 -14829.391} C_VEL
LIN {X 0,Y 334.365,Z 339.251,A -85,B 0,C 180,E1 -14829.868,E2 -14829.868} C_VEL
LIN {X 0,Y 332.825,Z 349.734,A -85,B 0,C 180,E1 -14831.055,E2 -14831.055} C_VEL
LIN {X 0,Y 331.106,Z 359.35,A -85,B 0,C 180,E1 -14832.395,E2 -14832.395} C_VEL
LIN {X 0,Y 329.716,Z 368.124,A -85,B 0,C 180,E1 -14833.913,E2 -14833.913} C_VEL
LIN {X 0,Y 328.308,Z 376.719,A -85,B 0,C 180,E1 -14835.749,E2 -14835.749} C_VEL
LIN {X 0,Y 326.963,Z 383.608,A -85,B 0,C 180,E1 -14837.588,E2 -14837.588} C_VEL
LIN {X 0,Y 326.122,Z 389.149,A -85,B 0,C 180,E1 -14839.445,E2 -14839.445} C_VEL
LIN {X 0,Y 325.519,Z 393.519,A -85,B 0,C 180,E1 -14841.308,E2 -14841.308} C_VEL
LIN {X 0,Y 325.204,Z 395.839,A -85,B 0,C 180,E1 -14842.55,E2 -14842.55} C_VEL
LIN {X 0,Y 324.98,Z 398.196,A -85,B 0,C 180,E1 -14844.16,E2 -14844.16} C_VEL
LIN {X 0,Y 324.878,Z 400.229,A -85,B 0,C 180,E1 -14846.279,E2 -14846.279} C_VEL
LIN {X 0,Y 324.835,Z 400.881,A -85,B 0,C 180,E1 -14847.52,E2 -14847.52} C_VEL
LIN {X 0,Y 324.823,Z 401.149,A -85,B 0,C 180,E1 -14848.76,E2 -14848.76} C_VEL
LIN {X 0,Y 324.877,Z 401.007,A -85,B 0,C 180,E1 -14850,E2 -14850} C_VEL
LIN {X 0,Y 324.84,Z 400.444,A -85,B 0,C 180,E1 -14851.24,E2 -14851.24} C_VEL
LIN {X 0,Y 324.848,Z 399.49,A -85,B 0,C 180,E1 -14852.48,E2 -14852.48} C_VEL
LIN {X 0,Y 324.906,Z 398.14,A -85,B 0,C 180,E1 -14853.721,E2 -14853.721} C_VEL
LIN {X 0,Y 324.988,Z 394.776,A -85,B 0,C 180,E1 -14855.855,E2 -14855.855} C_VEL
LIN {X 0,Y 325.239,Z 389.773,A -85,B 0,C 180,E1 -14858.074,E2 -14858.074} C_VEL
LIN {X 0,Y 325.795,Z 383.26,A -85,B 0,C 180,E1 -14860.251,E2 -14860.251} C_VEL
LIN {X 0,Y 326.449,Z 376.09,A -85,B 0,C 180,E1 -14862.117,E2 -14862.117} C_VEL
LIN {X 0,Y 327.448,Z 367.148,A -85,B 0,C 180,E1 -14863.972,E2 -14863.972} C_VEL
LIN {X 0,Y 328.327,Z 358.544,A -85,B 0,C 180,E1 -14865.424,E2 -14865.424} C_VEL
LIN {X 0,Y 329.42,Z 347.755,A -85,B 0,C 180,E1 -14866.898,E2 -14866.898} C_VEL
LIN {X 0,Y 330.667,Z 336.438,A -85,B 0,C 180,E1 -14868.109,E2 -14868.109} C_VEL
LIN {X 0,Y 330.723,Z 331.316,A -85,B 0,C 180,E1 -14868.587,E2 -14868.587} C_VEL
LIN {X 0,Y 329.381,Z 318.808,A -85,B 0,C 180,E1 -14869.62,E2 -14869.62} C_VEL
LIN {X 0,Y 327.58,Z 305.889,A -85,B 0,C 180,E1 -14870.431,E2 -14870.431} C_VEL
LIN {X 0,Y 325.662,Z 294.637,A -85,B 0,C 180,E1 -14870.983,E2 -14870.983} C_VEL
LIN {X 0,Y 326.038,Z 289.467,A -85,B 0,C 180,E1 -14874.177,E2 -14874.177} C_VEL
LIN {X 0,Y 326.565,Z 283.256,A -85,B 0,C 180,E1 -14878.069,E2 -14878.069} C_VEL
LIN {X 0,Y 327.216,Z 277.531,A -85,B 0,C 180,E1 -14881.749,E2 -14881.749} C_VEL
LIN {X 0,Y 327.732,Z 273.144,A -85,B 0,C 180,E1 -14884.629,E2 -14884.629} C_VEL
LIN {X 0,Y 327.792,Z 269.854,A -85,B 0,C 180,E1 -14886.893,E2 -14886.893} C_VEL
LIN {X 0,Y 327.132,Z 265.393,A -85,B 0,C 180,E1 -14890.128,E2 -14890.128} C_VEL
LIN {X 0,Y 326.639,Z 262.799,A -85,B 0,C 180,E1 -14892.25,E2 -14892.25} C_VEL
LIN {X 0,Y 326.548,Z 262.808,A -85,B 0,C 180,E1 -14896.471,E2 -14896.471} C_VEL
LIN {X 0,Y 326.552,Z 262.806,A -85,B 0,C 180,E1 -14899.784,E2 -14899.784} C_VEL
LIN {X 0,Y 326.623,Z 262.801,A -85,B 0,C 180,E1 -14902.951,E2 -14902.951} C_VEL
LIN {X 0,Y 326.604,Z 262.799,A -85,B 0,C 180,E1 -14905.979,E2 -14905.979} C_VEL
LIN {X 0,Y 326.609,Z 262.798,A -85,B 0,C 180,E1 -14909.396,E2 -14909.396} C_VEL
LIN {X 0,Y 326.609,Z 262.799,A -85,B 0,C 180,E1 -14913.134,E2 -14913.134} C_VEL
LIN {X 0,Y 326.627,Z 262.797,A -85,B 0,C 180,E1 -14915.868,E2 -14915.868} C_VEL
LIN {X 0,Y 326.65,Z 262.795,A -85,B 0,C 180,E1 -14919.863,E2 -14919.863} C_VEL
LIN {X 0,Y 326.695,Z 262.791,A -85,B 0,C 180,E1 -14922.47,E2 -14922.47} C_VEL
LIN {X 0,Y 326.754,Z 262.785,A -85,B 0,C 180,E1 -14926.313,E2 -14926.313} C_VEL
LIN {X 0,Y 326.8,Z 262.779,A -85,B 0,C 180,E1 -14930.092,E2 -14930.092} C_VEL
LIN {X 0,Y 326.983,Z 262.755,A -85,B 0,C 180,E1 -14933.829,E2 -14933.829} C_VEL
LIN {X 0,Y 327.04,Z 262.745,A -85,B 0,C 180,E1 -14937.535,E2 -14937.535} C_VEL
LIN {X 0,Y 327.211,Z 262.726,A -85,B 0,C 180,E1 -14939.999,E2 -14939.999} C_VEL
LIN {X 0,Y 327.041,Z 262.744,A -85,B 0,C 180,E1 -14942.462,E2 -14942.462} C_VEL
LIN {X 0,Y 326.963,Z 262.754,A -85,B 0,C 180,E1 -14946.683,E2 -14946.683} C_VEL
LIN {X 0,Y 326.805,Z 262.777,A -85,B 0,C 180,E1 -14949.905,E2 -14949.905} C_VEL
LIN {X 0,Y 326.75,Z 262.785,A -85,B 0,C 180,E1 -14953.684,E2 -14953.684} C_VEL
LIN {X 0,Y 326.69,Z 262.793,A -85,B 0,C 180,E1 -14957.527,E2 -14957.527} C_VEL
LIN {X 0,Y 326.656,Z 262.793,A -85,B 0,C 180,E1 -14960.134,E2 -14960.134} C_VEL
LIN {X 0,Y 326.642,Z 262.794,A -85,B 0,C 180,E1 -14964.128,E2 -14964.128} C_VEL
LIN {X 0,Y 326.675,Z 262.792,A -85,B 0,C 180,E1 -14966.857,E2 -14966.857} C_VEL
LIN {X 0,Y 326.629,Z 262.796,A -85,B 0,C 180,E1 -14970.61,E2 -14970.61} C_VEL
LIN {X 0,Y 326.596,Z 262.8,A -85,B 0,C 180,E1 -14974.019,E2 -14974.019} C_VEL
LIN {X 0,Y 326.618,Z 262.8,A -85,B 0,C 180,E1 -14977.238,E2 -14977.238} C_VEL
LIN {X 0,Y 326.624,Z 262.796,A -85,B 0,C 180,E1 -14980.202,E2 -14980.202} C_VEL
LIN {X 0,Y 326.607,Z 262.799,A -85,B 0,C 180,E1 -14983.515,E2 -14983.515} C_VEL
LIN {X 0,Y 326.575,Z 262.805,A -85,B 0,C 180,E1 -14987.026,E2 -14987.026} C_VEL
LIN {X 0,Y 326.601,Z 262.804,A -85,B 0,C 180,E1 -14990.772,E2 -14990.772} C_VEL
LIN {X 0,Y 326.602,Z 262.803,A -85,B 0,C 180,E1 -14994.48,E2 -14994.48} C_VEL
LIN {X 0,Y 326.596,Z 262.8,A -85,B 0,C 180,E1 -14997.455,E2 -14997.455} C_VEL
LIN {X 0,Y 326.635,Z 262.799,A -85,B 0,C 180,E1 -15000.339,E2 -15000.339} C_VEL
LIN {X 0,Y 326.638,Z 262.795,A -85,B 0,C 180,E1 -15003.139,E2 -15003.139} C_VEL
LIN {X 0,Y 326.536,Z 262.809,A -85,B 0,C 180,E1 -15005.863,E2 -15005.863} C_VEL
LIN {X 0,Y 326.459,Z 262.837,A -85,B 0,C 180,E1 -15008.155,E2 -15008.155} C_VEL
LIN {X 0,Y 326.319,Z 266.262,A -85,B 0,C 180,E1 -15011.37,E2 -15011.37} C_VEL
LIN {X 0,Y 326.057,Z 271.279,A -85,B 0,C 180,E1 -15015.911,E2 -15015.911} C_VEL
LIN {X 0,Y 325.768,Z 276.009,A -85,B 0,C 180,E1 -15020.062,E2 -15020.062} C_VEL
LIN {X 0,Y 325.746,Z 278.421,A -85,B 0,C 180,E1 -15022.149,E2 -15022.149} C_VEL
LIN {X 0,Y 328.51,Z 291.176,A -85,B 0,C 180,E1 -15022.819,E2 -15022.819} C_VEL
LIN {X 0,Y 330.721,Z 303.616,A -85,B 0,C 180,E1 -15023.691,E2 -15023.691} C_VEL
LIN {X 0,Y 331.696,Z 311.772,A -85,B 0,C 180,E1 -15024.376,E2 -15024.376} C_VEL
LIN {X 0,Y 330.737,Z 323.006,A -85,B 0,C 180,E1 -15025.43,E2 -15025.43} C_VEL
LIN {X 0,Y 329.54,Z 334.465,A -85,B 0,C 180,E1 -15026.791,E2 -15026.791} C_VEL
LIN {X 0,Y 328.537,Z 343.687,A -85,B 0,C 180,E1 -15028.161,E2 -15028.161} C_VEL
LIN {X 0,Y 327.615,Z 352.097,A -85,B 0,C 180,E1 -15029.693,E2 -15029.693} C_VEL
LIN {X 0,Y 326.594,Z 360.334,A -85,B 0,C 180,E1 -15031.541,E2 -15031.541} C_VEL
LIN {X 0,Y 326.067,Z 365.943,A -85,B 0,C 180,E1 -15033.089,E2 -15033.089} C_VEL
LIN {X 0,Y 325.554,Z 371.429,A -85,B 0,C 180,E1 -15034.954,E2 -15034.954} C_VEL
LIN {X 0,Y 325.333,Z 374.967,A -85,B 0,C 180,E1 -15036.446,E2 -15036.446} C_VEL
LIN {X 0,Y 324.929,Z 378.973,A -85,B 0,C 180,E1 -15038.708,E2 -15038.708} C_VEL
LIN {X 0,Y 324.766,Z 380.589,A -85,B 0,C 180,E1 -15039.969,E2 -15039.969} C_VEL
LIN {X 0,Y 324.74,Z 381.781,A -85,B 0,C 180,E1 -15041.231,E2 -15041.231} C_VEL
LIN {X 0,Y 324.757,Z 382.775,A -85,B 0,C 180,E1 -15043.145,E2 -15043.145} C_VEL
LIN {X 0,Y 324.737,Z 382.828,A -85,B 0,C 180,E1 -15045.052,E2 -15045.052} C_VEL
LIN {X 0,Y 324.861,Z 382.347,A -85,B 0,C 180,E1 -15046.334,E2 -15046.334} C_VEL
LIN {X 0,Y 325.119,Z 381.094,A -85,B 0,C 180,E1 -15047.992,E2 -15047.992} C_VEL
LIN {X 0,Y 325.587,Z 378.314,A -85,B 0,C 180,E1 -15050.204,E2 -15050.204} C_VEL
LIN {X 0,Y 326.248,Z 374.729,A -85,B 0,C 180,E1 -15052.14,E2 -15052.14} C_VEL
LIN {X 0,Y 327.1,Z 369.912,A -85,B 0,C 180,E1 -15054.093,E2 -15054.093} C_VEL
LIN {X 0,Y 328.384,Z 363.108,A -85,B 0,C 180,E1 -15056.213,E2 -15056.213} C_VEL
LIN {X 0,Y 329.666,Z 356,A -85,B 0,C 180,E1 -15057.969,E2 -15057.969} C_VEL
LIN {X 0,Y 331.123,Z 347.873,A -85,B 0,C 180,E1 -15059.596,E2 -15059.596} C_VEL
LIN {X 0,Y 332.748,Z 338.139,A -85,B 0,C 180,E1 -15061.162,E2 -15061.162} C_VEL
LIN {X 0,Y 334.329,Z 327.769,A -85,B 0,C 180,E1 -15062.5,E2 -15062.5} C_VEL
LIN {X 0,Y 335.83,Z 316.78,A -85,B 0,C 180,E1 -15063.627,E2 -15063.627} C_VEL
LIN {X 0,Y 334.473,Z 307.737,A -85,B 0,C 180,E1 -15064.563,E2 -15064.563} C_VEL
LIN {X 0,Y 331.612,Z 296.124,A -85,B 0,C 180,E1 -15065.651,E2 -15065.651} C_VEL
LIN {X 0,Y 327.631,Z 283.895,A -85,B 0,C 180,E1 -15066.643,E2 -15066.643} C_VEL
LIN {X 0,Y 326.014,Z 278.898,A -85,B 0,C 180,E1 -15067.019,E2 -15067.019} C_VEL
LIN {X 0,Y 326.285,Z 275.496,A -85,B 0,C 180,E1 -15070.253,E2 -15070.253} C_VEL
LIN {X 0,Y 326.59,Z 272.185,A -85,B 0,C 180,E1 -15073.519,E2 -15073.519} C_VEL
LIN {X 0,Y 326.952,Z 268.828,A -85,B 0,C 180,E1 -15076.956,E2 -15076.956} C_VEL
LIN {X 0,Y 326.959,Z 266.16,A -85,B 0,C 180,E1 -15079.848,E2 -15079.848} C_VEL
LIN {X 0,Y 326.681,Z 263.474,A -85,B 0,C 180,E1 -15082.962,E2 -15082.962} C_VEL
LIN {X 0,Y 326.608,Z 262.805,A -85,B 0,C 180,E1 -15084.852,E2 -15084.852} C_VEL
LIN {X 0,Y 326.596,Z 262.809,A -85,B 0,C 180,E1 -15087.456,E2 -15087.456} C_VEL
LIN {X 0,Y 326.623,Z 262.802,A -85,B 0,C 180,E1 -15089.344,E2 -15089.344} C_VEL
LIN {X 0,Y 326.043,Z 262.875,A -85,B 0,C 180,E1 -15090.373,E2 -15090.373} C_VEL
LIN {X 0,Y 323.22,Z 263.225,A -85,B 0,C 180,E1 -15092.048,E2 -15092.048} C_VEL
LIN {X 0,Y 320.765,Z 263.53,A -85,B 0,C 180,E1 -15093.405,E2 -15093.405} C_VEL
LIN {X 0,Y 319.695,Z 263.663,A -85,B 0,C 180,E1 -15094.455,E2 -15094.455} C_VEL
LIN {X 0,Y 319.603,Z 263.673,A -85,B 0,C 180,E1 -15094.812,E2 -15094.812} C_VEL
LIN {X 0,Y 319.596,Z 263.677,A -85,B 0,C 180,E1 -15098.05,E2 -15098.05} C_VEL
LIN {X 0,Y 319.682,Z 263.666,A -85,B 0,C 180,E1 -15100.962,E2 -15100.962} C_VEL
LIN {X 0,Y 319.722,Z 263.655,A -85,B 0,C 180,E1 -15105.277,E2 -15105.277} C_VEL
LIN {X 0,Y 319.743,Z 263.657,A -85,B 0,C 180,E1 -15109.874,E2 -15109.874} C_VEL
LIN {X 0,Y 319.904,Z 263.637,A -85,B 0,C 180,E1 -15112.427,E2 -15112.427} C_VEL
LIN {X 0,Y 319.738,Z 263.657,A -85,B 0,C 180,E1 -15114.957,E2 -15114.957} C_VEL
LIN {X 0,Y 319.984,Z 263.627,A -85,B 0,C 180,E1 -15117.484,E2 -15117.484} C_VEL
LIN {X 0,Y 320.122,Z 263.608,A -85,B 0,C 180,E1 -15120.002,E2 -15120.002} C_VEL
LIN {X 0,Y 319.984,Z 263.627,A -85,B 0,C 180,E1 -15122.519,E2 -15122.519} C_VEL
LIN {X 0,Y 319.943,Z 263.631,A -85,B 0,C 180,E1 -15126.307,E2 -15126.307} C_VEL
LIN {X 0,Y 319.837,Z 263.645,A -85,B 0,C 180,E1 -15128.85,E2 -15128.85} C_VEL
LIN {X 0,Y 319.676,Z 263.668,A -85,B 0,C 180,E1 -15132.701,E2 -15132.701} C_VEL
LIN {X 0,Y 319.694,Z 263.665,A -85,B 0,C 180,E1 -15135.297,E2 -15135.297} C_VEL
LIN {X 0,Y 319.67,Z 263.669,A -85,B 0,C 180,E1 -15139.257,E2 -15139.257} C_VEL
LIN {X 0,Y 319.565,Z 263.686,A -85,B 0,C 180,E1 -15143.321,E2 -15143.321} C_VEL
LIN {X 0,Y 319.579,Z 263.683,A -85,B 0,C 180,E1 -15146.094,E2 -15146.094} C_VEL
LIN {X 0,Y 319.556,Z 263.685,A -85,B 0,C 180,E1 -15148.938,E2 -15148.938} C_VEL
LIN {X 0,Y 319.522,Z 263.688,A -85,B 0,C 180,E1 -15151.864,E2 -15151.864} C_VEL
LIN {X 0,Y 319.578,Z 263.679,A -85,B 0,C 180,E1 -15155.544,E2 -15155.544} C_VEL
LIN {X 0,Y 319.556,Z 263.68,A -85,B 0,C 180,E1 -15158.012,E2 -15158.012} C_VEL
LIN {X 0,Y 319.537,Z 263.745,A -85,B 0,C 180,E1 -15161.288,E2 -15161.288} C_VEL
LIN {X 0,Y 320.255,Z 267.859,A -85,B 0,C 180,E1 -15165.394,E2 -15165.394} C_VEL
LIN {X 0,Y 320.923,Z 271.733,A -85,B 0,C 180,E1 -15168.931,E2 -15168.931} C_VEL
LIN {X 0,Y 321.484,Z 275.683,A -85,B 0,C 180,E1 -15172.259,E2 -15172.259} C_VEL
LIN {X 0,Y 321.533,Z 277.836,A -85,B 0,C 180,E1 -15173.975,E2 -15173.975} C_VEL
LIN {X 0,Y 321.118,Z 281.666,A -85,B 0,C 180,E1 -15176.829,E2 -15176.829} C_VEL
LIN {X 0,Y 320.309,Z 286.695,A -85,B 0,C 180,E1 -15180.418,E2 -15180.418} C_VEL
LIN {X 0,Y 319.575,Z 292.466,A -85,B 0,C 180,E1 -15184.379,E2 -15184.379} C_VEL
LIN {X 0,Y 319.418,Z 293.982,A -85,B 0,C 180,E1 -15185.402,E2 -15185.402} C_VEL
LIN {X 0,Y 322.037,Z 303.02,A -85,B 0,C 180,E1 -15186.022,E2 -15186.022} C_VEL
LIN {X 0,Y 325.02,Z 315.387,A -85,B 0,C 180,E1 -15187.004,E2 -15187.004} C_VEL
LIN {X 0,Y 327.084,Z 327.315,A -85,B 0,C 180,E1 -15188.11,E2 -15188.11} C_VEL
LIN {X 0,Y 327.883,Z 338.442,A -85,B 0,C 180,E1 -15189.289,E2 -15189.289} C_VEL
LIN {X 0,Y 326.133,Z 350.201,A -85,B 0,C 180,E1 -15190.651,E2 -15190.651} C_VEL
LIN {X 0,Y 324.355,Z 359.704,A -85,B 0,C 180,E1 -15192.016,E2 -15192.016} C_VEL
LIN {X 0,Y 322.885,Z 368.383,A -85,B 0,C 180,E1 -15193.563,E2 -15193.563} C_VEL
LIN {X 0,Y 321.672,Z 375.567,A -85,B 0,C 180,E1 -15195.125,E2 -15195.125} C_VEL
LIN {X 0,Y 320.252,Z 382.67,A -85,B 0,C 180,E1 -15197.001,E2 -15197.001} C_VEL
LIN {X 0,Y 319.125,Z 389.165,A -85,B 0,C 180,E1 -15199.211,E2 -15199.211} C_VEL
LIN {X 0,Y 318.465,Z 393.484,A -85,B 0,C 180,E1 -15201.114,E2 -15201.114} C_VEL
LIN {X 0,Y 318.147,Z 395.781,A -85,B 0,C 180,E1 -15202.384,E2 -15202.384} C_VEL
LIN {X 0,Y 317.867,Z 398.342,A -85,B 0,C 180,E1 -15204.245,E2 -15204.245} C_VEL
LIN {X 0,Y 317.788,Z 400.081,A -85,B 0,C 180,E1 -15206.196,E2 -15206.196} C_VEL
LIN {X 0,Y 317.756,Z 400.712,A -85,B 0,C 180,E1 -15207.465,E2 -15207.465} C_VEL
LIN {X 0,Y 317.735,Z 400.958,A -85,B 0,C 180,E1 -15208.733,E2 -15208.733} C_VEL
LIN {X 0,Y 317.784,Z 400.775,A -85,B 0,C 180,E1 -15210,E2 -15210} C_VEL
LIN {X 0,Y 317.751,Z 400.189,A -85,B 0,C 180,E1 -15211.267,E2 -15211.267} C_VEL
LIN {X 0,Y 317.769,Z 399.215,A -85,B 0,C 180,E1 -15212.535,E2 -15212.535} C_VEL
LIN {X 0,Y 317.814,Z 397.84,A -85,B 0,C 180,E1 -15213.804,E2 -15213.804} C_VEL
LIN {X 0,Y 317.881,Z 394.799,A -85,B 0,C 180,E1 -15215.78,E2 -15215.78} C_VEL
LIN {X 0,Y 318.067,Z 390.948,A -85,B 0,C 180,E1 -15217.618,E2 -15217.618} C_VEL
LIN {X 0,Y 318.558,Z 384.822,A -85,B 0,C 180,E1 -15219.845,E2 -15219.845} C_VEL
LIN {X 0,Y 319.192,Z 378.104,A -85,B 0,C 180,E1 -15221.751,E2 -15221.751} C_VEL
LIN {X 0,Y 320.195,Z 369.763,A -85,B 0,C 180,E1 -15223.648,E2 -15223.648} C_VEL
LIN {X 0,Y 321.256,Z 360.03,A -85,B 0,C 180,E1 -15225.408,E2 -15225.408} C_VEL
LIN {X 0,Y 322.326,Z 349.353,A -85,B 0,C 180,E1 -15226.955,E2 -15226.955} C_VEL
LIN {X 0,Y 323.525,Z 338.555,A -85,B 0,C 180,E1 -15228.196,E2 -15228.196} C_VEL
LIN {X 0,Y 323.936,Z 333.755,A -85,B 0,C 180,E1 -15228.663,E2 -15228.663} C_VEL
LIN {X 0,Y 322.667,Z 321.348,A -85,B 0,C 180,E1 -15229.76,E2 -15229.76} C_VEL
LIN {X 0,Y 320.909,Z 307.85,A -85,B 0,C 180,E1 -15230.679,E2 -15230.679} C_VEL
LIN {X 0,Y 318.623,Z 294.5,A -85,B 0,C 180,E1 -15231.342,E2 -15231.342} C_VEL
LIN {X 0,Y 319.137,Z 288,A -85,B 0,C 180,E1 -15235.456,E2 -15235.456} C_VEL
LIN {X 0,Y 319.766,Z 281.54,A -85,B 0,C 180,E1 -15239.637,E2 -15239.637} C_VEL
LIN {X 0,Y 320.486,Z 275.637,A -85,B 0,C 180,E1 -15243.558,E2 -15243.558} C_VEL
LIN {X 0,Y 320.815,Z 271.726,A -85,B 0,C 180,E1 -15246.261,E2 -15246.261} C_VEL
LIN {X 0,Y 320.404,Z 268.397,A -85,B 0,C 180,E1 -15248.691,E2 -15248.691} C_VEL
LIN {X 0,Y 319.582,Z 263.678,A -85,B 0,C 180,E1 -15252.359,E2 -15252.359} C_VEL
LIN {X 0,Y 319.511,Z 263.688,A -85,B 0,C 180,E1 -15257.008,E2 -15257.008} C_VEL
LIN {X 0,Y 319.514,Z 263.685,A -85,B 0,C 180,E1 -15260.364,E2 -15260.364} C_VEL
LIN {X 0,Y 319.576,Z 263.678,A -85,B 0,C 180,E1 -15264.456,E2 -15264.456} C_VEL
LIN {X 0,Y 319.522,Z 263.682,A -85,B 0,C 180,E1 -15268.136,E2 -15268.136} C_VEL
LIN {X 0,Y 319.568,Z 263.675,A -85,B 0,C 180,E1 -15271.602,E2 -15271.602} C_VEL
LIN {X 0,Y 319.569,Z 263.675,A -85,B 0,C 180,E1 -15275.3,E2 -15275.3} C_VEL
LIN {X 0,Y 319.562,Z 263.678,A -85,B 0,C 180,E1 -15278.044,E2 -15278.044} C_VEL
LIN {X 0,Y 319.685,Z 263.661,A -85,B 0,C 180,E1 -15280.961,E2 -15280.961} C_VEL
LIN {X 0,Y 319.726,Z 263.656,A -85,B 0,C 180,E1 -15285.274,E2 -15285.274} C_VEL
LIN {X 0,Y 319.747,Z 263.655,A -85,B 0,C 180,E1 -15289.871,E2 -15289.871} C_VEL
LIN {X 0,Y 319.907,Z 263.636,A -85,B 0,C 180,E1 -15292.424,E2 -15292.424} C_VEL
LIN {X 0,Y 319.738,Z 263.654,A -85,B 0,C 180,E1 -15294.954,E2 -15294.954} C_VEL
LIN {X 0,Y 319.983,Z 263.623,A -85,B 0,C 180,E1 -15297.481,E2 -15297.481} C_VEL
LIN {X 0,Y 320.162,Z 263.603,A -85,B 0,C 180,E1 -15299.998,E2 -15299.998} C_VEL
LIN {X 0,Y 319.985,Z 263.623,A -85,B 0,C 180,E1 -15302.516,E2 -15302.516} C_VEL
LIN {X 0,Y 319.922,Z 263.631,A -85,B 0,C 180,E1 -15306.674,E2 -15306.674} C_VEL
LIN {X 0,Y 319.75,Z 263.654,A -85,B 0,C 180,E1 -15310.126,E2 -15310.126} C_VEL
LIN {X 0,Y 319.722,Z 263.656,A -85,B 0,C 180,E1 -15314.723,E2 -15314.723} C_VEL
LIN {X 0,Y 319.68,Z 263.663,A -85,B 0,C 180,E1 -15319.036,E2 -15319.036} C_VEL
LIN {X 0,Y 319.56,Z 263.681,A -85,B 0,C 180,E1 -15323.318,E2 -15323.318} C_VEL
LIN {X 0,Y 319.625,Z 263.668,A -85,B 0,C 180,E1 -15326.087,E2 -15326.087} C_VEL
LIN {X 0,Y 319.58,Z 263.676,A -85,B 0,C 180,E1 -15328.933,E2 -15328.933} C_VEL
LIN {X 0,Y 319.522,Z 263.681,A -85,B 0,C 180,E1 -15331.861,E2 -15331.861} C_VEL
LIN {X 0,Y 319.569,Z 263.676,A -85,B 0,C 180,E1 -15335.542,E2 -15335.542} C_VEL
LIN {X 0,Y 319.573,Z 263.674,A -85,B 0,C 180,E1 -15338.006,E2 -15338.006} C_VEL
LIN {X 0,Y 319.585,Z 263.673,A -85,B 0,C 180,E1 -15341.61,E2 -15341.61} C_VEL
LIN {X 0,Y 319.552,Z 263.679,A -85,B 0,C 180,E1 -15345.27,E2 -15345.27} C_VEL
LIN {X 0,Y 319.518,Z 263.686,A -85,B 0,C 180,E1 -15348.711,E2 -15348.711} C_VEL
LIN {X 0,Y 319.567,Z 263.678,A -85,B 0,C 180,E1 -15352.343,E2 -15352.343} C_VEL
LIN {X 0,Y 319.549,Z 263.679,A -85,B 0,C 180,E1 -15355.123,E2 -15355.123} C_VEL
LIN {X 0,Y 319.555,Z 263.678,A -85,B 0,C 180,E1 -15359.059,E2 -15359.059} C_VEL
LIN {X 0,Y 319.576,Z 263.679,A -85,B 0,C 180,E1 -15362.496,E2 -15362.496} C_VEL
LIN {X 0,Y 319.512,Z 263.683,A -85,B 0,C 180,E1 -15365.297,E2 -15365.297} C_VEL
LIN {X 0,Y 319.428,Z 263.798,A -85,B 0,C 180,E1 -15368.206,E2 -15368.206} C_VEL
LIN {X 0,Y 319.19,Z 267.835,A -85,B 0,C 180,E1 -15372.046,E2 -15372.046} C_VEL
LIN {X 0,Y 318.986,Z 272.104,A -85,B 0,C 180,E1 -15375.975,E2 -15375.975} C_VEL
LIN {X 0,Y 318.706,Z 276.435,A -85,B 0,C 180,E1 -15379.839,E2 -15379.839} C_VEL
LIN {X 0,Y 318.671,Z 278.612,A -85,B 0,C 180,E1 -15381.749,E2 -15381.749} C_VEL
LIN {X 0,Y 321.62,Z 291.92,A -85,B 0,C 180,E1 -15382.492,E2 -15382.492} C_VEL
LIN {X 0,Y 323.864,Z 304.685,A -85,B 0,C 180,E1 -15383.418,E2 -15383.418} C_VEL
LIN {X 0,Y 324.794,Z 312.482,A -85,B 0,C 180,E1 -15384.101,E2 -15384.101} C_VEL
LIN {X 0,Y 323.821,Z 323.617,A -85,B 0,C 180,E1 -15385.176,E2 -15385.176} C_VEL
LIN {X 0,Y 322.585,Z 335.004,A -85,B 0,C 180,E1 -15386.565,E2 -15386.565} C_VEL
LIN {X 0,Y 321.433,Z 345.044,A -85,B 0,C 180,E1 -15388.121,E2 -15388.121} C_VEL
LIN {X 0,Y 320.502,Z 353.258,A -85,B 0,C 180,E1 -15389.686,E2 -15389.686} C_VEL
LIN {X 0,Y 319.482,Z 361.331,A -85,B 0,C 180,E1 -15391.576,E2 -15391.576} C_VEL
LIN {X 0,Y 318.944,Z 366.797,A -85,B 0,C 180,E1 -15393.158,E2 -15393.158} C_VEL
LIN {X 0,Y 318.461,Z 372.151,A -85,B 0,C 180,E1 -15395.064,E2 -15395.064} C_VEL
LIN {X 0,Y 318.146,Z 376.209,A -85,B 0,C 180,E1 -15396.915,E2 -15396.915} C_VEL
LIN {X 0,Y 317.804,Z 379.467,A -85,B 0,C 180,E1 -15398.905,E2 -15398.905} C_VEL
LIN {X 0,Y 317.654,Z 381.026,A -85,B 0,C 180,E1 -15400.195,E2 -15400.195} C_VEL
LIN {X 0,Y 317.658,Z 382.116,A -85,B 0,C 180,E1 -15401.485,E2 -15401.485} C_VEL
LIN {X 0,Y 317.679,Z 382.981,A -85,B 0,C 180,E1 -15403.252,E2 -15403.252} C_VEL
LIN {X 0,Y 317.68,Z 382.986,A -85,B 0,C 180,E1 -15405.395,E2 -15405.395} C_VEL
LIN {X 0,Y 317.815,Z 382.417,A -85,B 0,C 180,E1 -15406.706,E2 -15406.706} C_VEL
LIN {X 0,Y 318.051,Z 381.314,A -85,B 0,C 180,E1 -15408.169,E2 -15408.169} C_VEL
LIN {X 0,Y 318.283,Z 380.051,A -85,B 0,C 180,E1 -15409.342,E2 -15409.342} C_VEL
LIN {X 0,Y 318.855,Z 377.068,A -85,B 0,C 180,E1 -15411.326,E2 -15411.326} C_VEL
LIN {X 0,Y 319.652,Z 372.965,A -85,B 0,C 180,E1 -15413.312,E2 -15413.312} C_VEL
LIN {X 0,Y 320.895,Z 366.546,A -85,B 0,C 180,E1 -15415.629,E2 -15415.629} C_VEL
LIN {X 0,Y 322.32,Z 359.484,A -85,B 0,C 180,E1 -15417.602,E2 -15417.602} C_VEL
LIN {X 0,Y 323.721,Z 352.2,A -85,B 0,C 180,E1 -15419.24,E2 -15419.24} C_VEL
LIN {X 0,Y 325.329,Z 343.285,A -85,B 0,C 180,E1 -15420.867,E2 -15420.867} C_VEL
LIN {X 0,Y 326.98,Z 333.404,A -85,B 0,C 180,E1 -15422.32,E2 -15422.32} C_VEL
LIN {X 0,Y 328.589,Z 322.62,A -85,B 0,C 180,E1 -15423.59,E2 -15423.59} C_VEL
LIN {X 0,Y 329.279,Z 317.434,A -85,B 0,C 180,E1 -15424.103,E2 -15424.103} C_VEL
LIN {X 0,Y 327.661,Z 308.096,A -85,B 0,C 180,E1 -15425.122,E2 -15425.122} C_VEL
LIN {X 0,Y 324.709,Z 296.248,A -85,B 0,C 180,E1 -15426.273,E2 -15426.273} C_VEL
LIN {X 0,Y 320.568,Z 283.737,A -85,B 0,C 180,E1 -15427.329,E2 -15427.329} C_VEL
LIN {X 0,Y 319.06,Z 279.447,A -85,B 0,C 180,E1 -15427.647,E2 -15427.647} C_VEL
LIN {X 0,Y 319.025,Z 279.047,A -85,B 0,C 180,E1 -15427.748,E2 -15427.748} C_VEL
LIN {X 0,Y 319.377,Z 275.156,A -85,B 0,C 180,E1 -15431.57,E2 -15431.57} C_VEL
LIN {X 0,Y 319.798,Z 271.503,A -85,B 0,C 180,E1 -15435.315,E2 -15435.315} C_VEL
LIN {X 0,Y 319.964,Z 268.702,A -85,B 0,C 180,E1 -15438.313,E2 -15438.313} C_VEL
LIN {X 0,Y 319.908,Z 266.826,A -85,B 0,C 180,E1 -15440.427,E2 -15440.427} C_VEL
LIN {X 0,Y 319.605,Z 264.205,A -85,B 0,C 180,E1 -15443.581,E2 -15443.581} C_VEL
LIN {X 0,Y 319.569,Z 263.683,A -85,B 0,C 180,E1 -15444.458,E2 -15444.458} C_VEL
LIN {X 0,Y 319.521,Z 263.688,A -85,B 0,C 180,E1 -15448.139,E2 -15448.139} C_VEL
LIN {X 0,Y 319.606,Z 263.674,A -85,B 0,C 180,E1 -15451.59,E2 -15451.59} C_VEL
LIN {X 0,Y 319.603,Z 263.673,A -85,B 0,C 180,E1 -15454.812,E2 -15454.812} C_VEL
LIN {X 0,Y 318.921,Z 263.76,A -85,B 0,C 180,E1 -15455.863,E2 -15455.863} C_VEL
LIN {X 0,Y 316.065,Z 264.113,A -85,B 0,C 180,E1 -15457.574,E2 -15457.574} C_VEL
LIN {X 0,Y 313.673,Z 264.413,A -85,B 0,C 180,E1 -15458.961,E2 -15458.961} C_VEL
LIN {X 0,Y 312.673,Z 264.536,A -85,B 0,C 180,E1 -15460.034,E2 -15460.034} C_VEL
LIN {X 0,Y 312.605,Z 264.545,A -85,B 0,C 180,E1 -15460.398,E2 -15460.398} C_VEL
LIN {X 0,Y 312.629,Z 264.542,A -85,B 0,C 180,E1 -15464.352,E2 -15464.352} C_VEL
LIN {X 0,Y 312.625,Z 264.545,A -85,B 0,C 180,E1 -15467.01,E2 -15467.01} C_VEL
LIN {X 0,Y 312.819,Z 264.52,A -85,B 0,C 180,E1 -15471.305,E2 -15471.305} C_VEL
LIN {X 0,Y 312.892,Z 264.509,A -85,B 0,C 180,E1 -15473.553,E2 -15473.553} C_VEL
LIN {X 0,Y 312.93,Z 264.505,A -85,B 0,C 180,E1 -15477.427,E2 -15477.427} C_VEL
LIN {X 0,Y 313.075,Z 264.486,A -85,B 0,C 180,E1 -15480.002,E2 -15480.002} C_VEL
LIN {X 0,Y 312.93,Z 264.506,A -85,B 0,C 180,E1 -15482.576,E2 -15482.576} C_VEL
LIN {X 0,Y 312.902,Z 264.509,A -85,B 0,C 180,E1 -15486.45,E2 -15486.45} C_VEL
LIN {X 0,Y 312.782,Z 264.525,A -85,B 0,C 180,E1 -15489.051,E2 -15489.051} C_VEL
LIN {X 0,Y 312.629,Z 264.544,A -85,B 0,C 180,E1 -15492.993,E2 -15492.993} C_VEL
LIN {X 0,Y 312.633,Z 264.545,A -85,B 0,C 180,E1 -15495.651,E2 -15495.651} C_VEL
LIN {X 0,Y 312.626,Z 264.547,A -85,B 0,C 180,E1 -15499.238,E2 -15499.238} C_VEL
LIN {X 0,Y 312.541,Z 264.559,A -85,B 0,C 180,E1 -15502.79,E2 -15502.79} C_VEL
LIN {X 0,Y 312.562,Z 264.557,A -85,B 0,C 180,E1 -15505.923,E2 -15505.923} C_VEL
LIN {X 0,Y 312.501,Z 264.564,A -85,B 0,C 180,E1 -15509.656,E2 -15509.656} C_VEL
LIN {X 0,Y 312.518,Z 264.558,A -85,B 0,C 180,E1 -15513.69,E2 -15513.69} C_VEL
LIN {X 0,Y 312.524,Z 264.556,A -85,B 0,C 180,E1 -15517.387,E2 -15517.387} C_VEL
LIN {X 0,Y 312.525,Z 264.688,A -85,B 0,C 180,E1 -15520.705,E2 -15520.705} C_VEL
LIN {X 0,Y 313.059,Z 267.956,A -85,B 0,C 180,E1 -15524.103,E2 -15524.103} C_VEL
LIN {X 0,Y 313.759,Z 271.795,A -85,B 0,C 180,E1 -15527.781,E2 -15527.781} C_VEL
LIN {X 0,Y 314.342,Z 276,A -85,B 0,C 180,E1 -15531.494,E2 -15531.494} C_VEL
LIN {X 0,Y 314.521,Z 278.495,A -85,B 0,C 180,E1 -15533.556,E2 -15533.556} C_VEL
LIN {X 0,Y 314.111,Z 282.661,A -85,B 0,C 180,E1 -15536.759,E2 -15536.759} C_VEL
LIN {X 0,Y 313.266,Z 287.693,A -85,B 0,C 180,E1 -15540.426,E2 -15540.426} C_VEL
LIN {X 0,Y 312.575,Z 292.875,A -85,B 0,C 180,E1 -15544.077,E2 -15544.077} C_VEL
LIN {X 0,Y 312.452,Z 293.778,A -85,B 0,C 180,E1 -15544.7,E2 -15544.7} C_VEL
LIN {X 0,Y 314.313,Z 300.015,A -85,B 0,C 180,E1 -15545.132,E2 -15545.132} C_VEL
LIN {X 0,Y 317.479,Z 311.718,A -85,B 0,C 180,E1 -15546.067,E2 -15546.067} C_VEL
LIN {X 0,Y 319.738,Z 323.241,A -85,B 0,C 180,E1 -15547.126,E2 -15547.126} C_VEL
LIN {X 0,Y 321.056,Z 334.551,A -85,B 0,C 180,E1 -15548.322,E2 -15548.322} C_VEL
LIN {X 0,Y 321.144,Z 340.467,A -85,B 0,C 180,E1 -15549.001,E2 -15549.001} C_VEL
LIN {X 0,Y 319.229,Z 351.835,A -85,B 0,C 180,E1 -15550.383,E2 -15550.383} C_VEL
LIN {X 0,Y 317.288,Z 361.906,A -85,B 0,C 180,E1 -15551.935,E2 -15551.935} C_VEL
LIN {X 0,Y 315.858,Z 370.144,A -85,B 0,C 180,E1 -15553.52,E2 -15553.52} C_VEL
LIN {X 0,Y 314.278,Z 378.237,A -85,B 0,C 180,E1 -15555.43,E2 -15555.43} C_VEL
LIN {X 0,Y 313.085,Z 383.769,A -85,B 0,C 180,E1 -15557.028,E2 -15557.028} C_VEL
LIN {X 0,Y 312.122,Z 389.193,A -85,B 0,C 180,E1 -15558.966,E2 -15558.966} C_VEL
LIN {X 0,Y 311.43,Z 393.458,A -85,B 0,C 180,E1 -15560.911,E2 -15560.911} C_VEL
LIN {X 0,Y 311.08,Z 395.728,A -85,B 0,C 180,E1 -15562.21,E2 -15562.21} C_VEL
LIN {X 0,Y 310.77,Z 398.459,A -85,B 0,C 180,E1 -15564.306,E2 -15564.306} C_VEL
LIN {X 0,Y 310.702,Z 399.935,A -85,B 0,C 180,E1 -15566.109,E2 -15566.109} C_VEL
LIN {X 0,Y 310.679,Z 400.545,A -85,B 0,C 180,E1 -15567.407,E2 -15567.407} C_VEL
LIN {X 0,Y 310.65,Z 400.757,A -85,B 0,C 180,E1 -15568.704,E2 -15568.704} C_VEL
LIN {X 0,Y 310.694,Z 400.542,A -85,B 0,C 180,E1 -15570,E2 -15570} C_VEL
LIN {X 0,Y 310.665,Z 399.936,A -85,B 0,C 180,E1 -15571.296,E2 -15571.296} C_VEL
LIN {X 0,Y 310.692,Z 398.94,A -85,B 0,C 180,E1 -15572.593,E2 -15572.593} C_VEL
LIN {X 0,Y 310.726,Z 397.531,A -85,B 0,C 180,E1 -15573.891,E2 -15573.891} C_VEL
LIN {X 0,Y 310.806,Z 394.709,A -85,B 0,C 180,E1 -15575.759,E2 -15575.759} C_VEL
LIN {X 0,Y 311.009,Z 390.551,A -85,B 0,C 180,E1 -15577.792,E2 -15577.792} C_VEL
LIN {X 0,Y 311.535,Z 384.346,A -85,B 0,C 180,E1 -15580.069,E2 -15580.069} C_VEL
LIN {X 0,Y 312.205,Z 377.563,A -85,B 0,C 180,E1 -15582.018,E2 -15582.018} C_VEL
LIN {X 0,Y 313.237,Z 369.136,A -85,B 0,C 180,E1 -15583.957,E2 -15583.957} C_VEL
LIN {X 0,Y 314.233,Z 360.426,A -85,B 0,C 180,E1 -15585.568,E2 -15585.568} C_VEL
LIN {X 0,Y 315.351,Z 349.672,A -85,B 0,C 180,E1 -15587.175,E2 -15587.175} C_VEL
LIN {X 0,Y 316.569,Z 339.001,A -85,B 0,C 180,E1 -15588.442,E2 -15588.442} C_VEL
LIN {X 0,Y 316.979,Z 334.255,A -85,B 0,C 180,E1 -15588.921,E2 -15588.921} C_VEL
LIN {X 0,Y 315.724,Z 321.671,A -85,B 0,C 180,E1 -15590.075,E2 -15590.075} C_VEL
LIN {X 0,Y 313.987,Z 308.34,A -85,B 0,C 180,E1 -15591.018,E2 -15591.018} C_VEL
LIN {X 0,Y 311.582,Z 294.309,A -85,B 0,C 180,E1 -15591.745,E2 -15591.745} C_VEL
LIN {X 0,Y 312.105,Z 288.157,A -85,B 0,C 180,E1 -15595.744,E2 -15595.744} C_VEL
LIN {X 0,Y 312.83,Z 281.205,A -85,B 0,C 180,E1 -15600.363,E2 -15600.363} C_VEL
LIN {X 0,Y 313.541,Z 275.776,A -85,B 0,C 180,E1 -15604.081,E2 -15604.081} C_VEL
LIN {X 0,Y 313.795,Z 272.666,A -85,B 0,C 180,E1 -15606.264,E2 -15606.264} C_VEL
LIN {X 0,Y 313.332,Z 269.148,A -85,B 0,C 180,E1 -15608.904,E2 -15608.904} C_VEL
LIN {X 0,Y 312.54,Z 264.555,A -85,B 0,C 180,E1 -15612.531,E2 -15612.531} C_VEL
LIN {X 0,Y 312.45,Z 264.564,A -85,B 0,C 180,E1 -15616.035,E2 -15616.035} C_VEL
LIN {X 0,Y 312.452,Z 264.563,A -85,B 0,C 180,E1 -15619.885,E2 -15619.885} C_VEL
LIN {X 0,Y 312.531,Z 264.553,A -85,B 0,C 180,E1 -15624.05,E2 -15624.05} C_VEL
LIN {X 0,Y 312.499,Z 264.557,A -85,B 0,C 180,E1 -15627.332,E2 -15627.332} C_VEL
LIN {X 0,Y 312.503,Z 264.555,A -85,B 0,C 180,E1 -15631.29,E2 -15631.29} C_VEL
LIN {X 0,Y 312.543,Z 264.553,A -85,B 0,C 180,E1 -15634.706,E2 -15634.706} C_VEL
LIN {X 0,Y 312.53,Z 264.554,A -85,B 0,C 180,E1 -15638.911,E2 -15638.911} C_VEL
LIN {X 0,Y 312.634,Z 264.539,A -85,B 0,C 180,E1 -15641.655,E2 -15641.655} C_VEL
LIN {X 0,Y 312.689,Z 264.534,A -85,B 0,C 180,E1 -15645.685,E2 -15645.685} C_VEL
LIN {X 0,Y 312.693,Z 264.532,A -85,B 0,C 180,E1 -15649.64,E2 -15649.64} C_VEL
LIN {X 0,Y 312.848,Z 264.517,A -85,B 0,C 180,E1 -15652.252,E2 -15652.252} C_VEL
LIN {X 0,Y 312.708,Z 264.529,A -85,B 0,C 180,E1 -15654.841,E2 -15654.841} C_VEL
LIN {X 0,Y 312.986,Z 264.49,A -85,B 0,C 180,E1 -15658.712,E2 -15658.712} C_VEL
LIN {X 0,Y 313.113,Z 264.48,A -85,B 0,C 180,E1 -15659.998,E2 -15659.998} C_VEL
LIN {X 0,Y 312.931,Z 264.501,A -85,B 0,C 180,E1 -15662.573,E2 -15662.573} C_VEL
LIN {X 0,Y 312.885,Z 264.508,A -85,B 0,C 180,E1 -15666.658,E2 -15666.658} C_VEL
LIN {X 0,Y 312.78,Z 264.521,A -85,B 0,C 180,E1 -15669.048,E2 -15669.048} C_VEL
LIN {X 0,Y 312.625,Z 264.541,A -85,B 0,C 180,E1 -15672.99,E2 -15672.99} C_VEL
LIN {X 0,Y 312.629,Z 264.543,A -85,B 0,C 180,E1 -15675.648,E2 -15675.648} C_VEL
LIN {X 0,Y 312.621,Z 264.544,A -85,B 0,C 180,E1 -15679.235,E2 -15679.235} C_VEL
LIN {X 0,Y 312.536,Z 264.552,A -85,B 0,C 180,E1 -15682.788,E2 -15682.788} C_VEL
LIN {X 0,Y 312.593,Z 264.545,A -85,B 0,C 180,E1 -15685.934,E2 -15685.934} C_VEL
LIN {X 0,Y 312.535,Z 264.551,A -85,B 0,C 180,E1 -15689.649,E2 -15689.649} C_VEL
LIN {X 0,Y 312.509,Z 264.555,A -85,B 0,C 180,E1 -15693.688,E2 -15693.688} C_VEL
LIN {X 0,Y 312.531,Z 264.554,A -85,B 0,C 180,E1 -15697.382,E2 -15697.382} C_VEL
LIN {X 0,Y 312.515,Z 264.557,A -85,B 0,C 180,E1 -15700.703,E2 -15700.703} C_VEL
LIN {X 0,Y 312.519,Z 264.554,A -85,B 0,C 180,E1 -15704.195,E2 -15704.195} C_VEL
LIN {X 0,Y 312.476,Z 264.558,A -85,B 0,C 180,E1 -15707.917,E2 -15707.917} C_VEL
LIN {X 0,Y 312.495,Z 264.556,A -85,B 0,C 180,E1 -15711.917,E2 -15711.917} C_VEL
LIN {X 0,Y 312.522,Z 264.555,A -85,B 0,C 180,E1 -15714.22,E2 -15714.22} C_VEL
LIN {X 0,Y 312.492,Z 264.557,A -85,B 0,C 180,E1 -15717.333,E2 -15717.333} C_VEL
LIN {X 0,Y 312.53,Z 264.552,A -85,B 0,C 180,E1 -15721.28,E2 -15721.28} C_VEL
LIN {X 0,Y 312.518,Z 264.557,A -85,B 0,C 180,E1 -15724.706,E2 -15724.706} C_VEL
LIN {X 0,Y 312.375,Z 264.712,A -85,B 0,C 180,E1 -15728.209,E2 -15728.209} C_VEL
LIN {X 0,Y 312.185,Z 268.231,A -85,B 0,C 180,E1 -15731.629,E2 -15731.629} C_VEL
LIN {X 0,Y 311.943,Z 272.516,A -85,B 0,C 180,E1 -15735.651,E2 -15735.651} C_VEL
LIN {X 0,Y 311.657,Z 276.859,A -85,B 0,C 180,E1 -15739.607,E2 -15739.607} C_VEL
LIN {X 0,Y 311.607,Z 278.803,A -85,B 0,C 180,E1 -15741.358,E2 -15741.358} C_VEL
LIN {X 0,Y 314.671,Z 292.2,A -85,B 0,C 180,E1 -15742.121,E2 -15742.121} C_VEL
LIN {X 0,Y 316.932,Z 305.309,A -85,B 0,C 180,E1 -15743.1,E2 -15743.1} C_VEL
LIN {X 0,Y 317.879,Z 313.148,A -85,B 0,C 180,E1 -15743.813,E2 -15743.813} C_VEL
LIN {X 0,Y 316.896,Z 324.188,A -85,B 0,C 180,E1 -15744.911,E2 -15744.911} C_VEL
LIN {X 0,Y 315.615,Z 335.499,A -85,B 0,C 180,E1 -15746.329,E2 -15746.329} C_VEL
LIN {X 0,Y 314.565,Z 344.586,A -85,B 0,C 180,E1 -15747.759,E2 -15747.759} C_VEL
LIN {X 0,Y 313.582,Z 352.912,A -85,B 0,C 180,E1 -15749.358,E2 -15749.358} C_VEL
LIN {X 0,Y 312.484,Z 361.084,A -85,B 0,C 180,E1 -15751.289,E2 -15751.289} C_VEL
LIN {X 0,Y 311.821,Z 367.641,A -85,B 0,C 180,E1 -15753.23,E2 -15753.23} C_VEL
LIN {X 0,Y 311.369,Z 372.866,A -85,B 0,C 180,E1 -15755.18,E2 -15755.18} C_VEL
LIN {X 0,Y 311.002,Z 376.936,A -85,B 0,C 180,E1 -15757.139,E2 -15757.139} C_VEL
LIN {X 0,Y 310.698,Z 379.958,A -85,B 0,C 180,E1 -15759.11,E2 -15759.11} C_VEL
LIN {X 0,Y 310.546,Z 381.419,A -85,B 0,C 180,E1 -15760.431,E2 -15760.431} C_VEL
LIN {X 0,Y 310.55,Z 382.449,A -85,B 0,C 180,E1 -15761.752,E2 -15761.752} C_VEL
LIN {X 0,Y 310.574,Z 383.181,A -85,B 0,C 180,E1 -15763.341,E2 -15763.341} C_VEL
LIN {X 0,Y 310.606,Z 383.112,A -85,B 0,C 180,E1 -15765.754,E2 -15765.754} C_VEL
LIN {X 0,Y 310.798,Z 382.489,A -85,B 0,C 180,E1 -15767.095,E2 -15767.095} C_VEL
LIN {X 0,Y 311.02,Z 381.462,A -85,B 0,C 180,E1 -15768.442,E2 -15768.442} C_VEL
LIN {X 0,Y 311.316,Z 379.977,A -85,B 0,C 180,E1 -15769.793,E2 -15769.793} C_VEL
LIN {X 0,Y 311.958,Z 376.881,A -85,B 0,C 180,E1 -15771.821,E2 -15771.821} C_VEL
LIN {X 0,Y 312.818,Z 372.642,A -85,B 0,C 180,E1 -15773.853,E2 -15773.853} C_VEL
LIN {X 0,Y 314.195,Z 366.086,A -85,B 0,C 180,E1 -15776.216,E2 -15776.216} C_VEL
LIN {X 0,Y 315.68,Z 358.835,A -85,B 0,C 180,E1 -15778.234,E2 -15778.234} C_VEL
LIN {X 0,Y 317.473,Z 349.897,A -85,B 0,C 180,E1 -15780.187,E2 -15780.187} C_VEL
LIN {X 0,Y 319.319,Z 340.159,A -85,B 0,C 180,E1 -15781.885,E2 -15781.885} C_VEL
LIN {X 0,Y 321.166,Z 329.23,A -85,B 0,C 180,E1 -15783.384,E2 -15783.384} C_VEL
LIN {X 0,Y 322.685,Z 319.116,A -85,B 0,C 180,E1 -15784.49,E2 -15784.49} C_VEL
LIN {X 0,Y 321.026,Z 309.056,A -85,B 0,C 180,E1 -15785.641,E2 -15785.641} C_VEL
LIN {X 0,Y 318.18,Z 297.689,A -85,B 0,C 180,E1 -15786.801,E2 -15786.801} C_VEL
LIN {X 0,Y 314.298,Z 285.763,A -85,B 0,C 180,E1 -15787.874,E2 -15787.874} C_VEL
LIN {X 0,Y 312.108,Z 279.88,A -85,B 0,C 180,E1 -15788.346,E2 -15788.346} C_VEL
LIN {X 0,Y 312.045,Z 279.315,A -85,B 0,C 180,E1 -15788.418,E2 -15788.418} C_VEL
LIN {X 0,Y 312.416,Z 275.33,A -85,B 0,C 180,E1 -15792.443,E2 -15792.443} C_VEL
LIN {X 0,Y 312.85,Z 271.978,A -85,B 0,C 180,E1 -15795.959,E2 -15795.959} C_VEL
LIN {X 0,Y 312.926,Z 268.937,A -85,B 0,C 180,E1 -15799.362,E2 -15799.362} C_VEL
LIN {X 0,Y 312.721,Z 266.193,A -85,B 0,C 180,E1 -15802.645,E2 -15802.645} C_VEL
LIN {X 0,Y 312.56,Z 264.94,A -85,B 0,C 180,E1 -15804.226,E2 -15804.226} C_VEL
LIN {X 0,Y 312.508,Z 264.564,A -85,B 0,C 180,E1 -15806.312,E2 -15806.312} C_VEL
LIN {X 0,Y 312.534,Z 264.558,A -85,B 0,C 180,E1 -15810.351,E2 -15810.351} C_VEL
LIN {X 0,Y 312.594,Z 264.548,A -85,B 0,C 180,E1 -15814.065,E2 -15814.065} C_VEL
LIN {X 0,Y 312.581,Z 264.547,A -85,B 0,C 180,E1 -15817.53,E2 -15817.53} C_VEL
LIN {X 0,Y 312.605,Z 264.545,A -85,B 0,C 180,E1 -15820.398,E2 -15820.398} C_VEL
LIN {X 0,Y 311.98,Z 264.625,A -85,B 0,C 180,E1 -15821.474,E2 -15821.474} C_VEL
LIN {X 0,Y 309.16,Z 264.974,A -85,B 0,C 180,E1 -15823.226,E2 -15823.226} C_VEL
LIN {X 0,Y 306.735,Z 265.276,A -85,B 0,C 180,E1 -15824.646,E2 -15824.646} C_VEL
LIN {X 0,Y 305.678,Z 265.404,A -85,B 0,C 180,E1 -15825.746,E2 -15825.746} C_VEL
LIN {X 0,Y 305.585,Z 265.415,A -85,B 0,C 180,E1 -15826.118,E2 -15826.118} C_VEL
LIN {X 0,Y 305.627,Z 265.416,A -85,B 0,C 180,E1 -15829.401,E2 -15829.401} C_VEL
LIN {X 0,Y 305.788,Z 265.395,A -85,B 0,C 180,E1 -15832.075,E2 -15832.075} C_VEL
LIN {X 0,Y 305.679,Z 265.41,A -85,B 0,C 180,E1 -15834.725,E2 -15834.725} C_VEL
LIN {X 0,Y 305.949,Z 265.376,A -85,B 0,C 180,E1 -15838.685,E2 -15838.685} C_VEL
LIN {X 0,Y 305.948,Z 265.375,A -85,B 0,C 180,E1 -15841.318,E2 -15841.318} C_VEL
LIN {X 0,Y 305.682,Z 265.408,A -85,B 0,C 180,E1 -15845.278,E2 -15845.278} C_VEL
LIN {X 0,Y 305.807,Z 265.392,A -85,B 0,C 180,E1 -15847.927,E2 -15847.927} C_VEL
LIN {X 0,Y 305.598,Z 265.418,A -85,B 0,C 180,E1 -15851.947,E2 -15851.947} C_VEL
LIN {X 0,Y 305.633,Z 265.417,A -85,B 0,C 180,E1 -15855.036,E2 -15855.036} C_VEL
LIN {X 0,Y 305.573,Z 265.426,A -85,B 0,C 180,E1 -15859.447,E2 -15859.447} C_VEL
LIN {X 0,Y 305.485,Z 265.439,A -85,B 0,C 180,E1 -15863.042,E2 -15863.042} C_VEL
LIN {X 0,Y 305.494,Z 265.437,A -85,B 0,C 180,E1 -15866.209,E2 -15866.209} C_VEL
LIN {X 0,Y 305.461,Z 265.441,A -85,B 0,C 180,E1 -15869.041,E2 -15869.041} C_VEL
LIN {X 0,Y 305.434,Z 265.442,A -85,B 0,C 180,E1 -15871.955,E2 -15871.955} C_VEL
LIN {X 0,Y 305.461,Z 265.436,A -85,B 0,C 180,E1 -15875.115,E2 -15875.115} C_VEL
LIN {X 0,Y 305.472,Z 265.434,A -85,B 0,C 180,E1 -15879.257,E2 -15879.257} C_VEL
LIN {X 0,Y 305.519,Z 265.643,A -85,B 0,C 180,E1 -15880.1,E2 -15880.1} C_VEL
LIN {X 0,Y 306.174,Z 269.917,A -85,B 0,C 180,E1 -15884.638,E2 -15884.638} C_VEL
LIN {X 0,Y 306.862,Z 273.789,A -85,B 0,C 180,E1 -15888.382,E2 -15888.382} C_VEL
LIN {X 0,Y 307.386,Z 277.691,A -85,B 0,C 180,E1 -15891.88,E2 -15891.88} C_VEL
LIN {X 0,Y 307.512,Z 279.676,A -85,B 0,C 180,E1 -15893.544,E2 -15893.544} C_VEL
LIN {X 0,Y 307.106,Z 283.657,A -85,B 0,C 180,E1 -15896.687,E2 -15896.687} C_VEL
LIN {X 0,Y 306.151,Z 289.084,A -85,B 0,C 180,E1 -15900.732,E2 -15900.732} C_VEL
LIN {X 0,Y 305.565,Z 293.732,A -85,B 0,C 180,E1 -15903.97,E2 -15903.97} C_VEL
LIN {X 0,Y 307.508,Z 300.148,A -85,B 0,C 180,E1 -15904.436,E2 -15904.436} C_VEL
LIN {X 0,Y 310.987,Z 312.863,A -85,B 0,C 180,E1 -15905.516,E2 -15905.516} C_VEL
LIN {X 0,Y 313.119,Z 324.074,A -85,B 0,C 180,E1 -15906.598,E2 -15906.598} C_VEL
LIN {X 0,Y 314.426,Z 335.301,A -85,B 0,C 180,E1 -15907.841,E2 -15907.841} C_VEL
LIN {X 0,Y 314.559,Z 341.105,A -85,B 0,C 180,E1 -15908.54,E2 -15908.54} C_VEL
LIN {X 0,Y 312.588,Z 352.295,A -85,B 0,C 180,E1 -15909.949,E2 -15909.949} C_VEL
LIN {X 0,Y 310.548,Z 362.219,A -85,B 0,C 180,E1 -15911.529,E2 -15911.529} C_VEL
LIN {X 0,Y 309.027,Z 370.367,A -85,B 0,C 180,E1 -15913.145,E2 -15913.145} C_VEL
LIN {X 0,Y 307.406,Z 378.387,A -85,B 0,C 180,E1 -15915.096,E2 -15915.096} C_VEL
LIN {X 0,Y 306.156,Z 383.855,A -85,B 0,C 180,E1 -15916.729,E2 -15916.729} C_VEL
LIN {X 0,Y 305.131,Z 389.223,A -85,B 0,C 180,E1 -15918.71,E2 -15918.71} C_VEL
LIN {X 0,Y 304.413,Z 393.434,A -85,B 0,C 180,E1 -15920.7,E2 -15920.7} C_VEL
LIN {X 0,Y 304.035,Z 395.679,A -85,B 0,C 180,E1 -15922.028,E2 -15922.028} C_VEL
LIN {X 0,Y 303.664,Z 398.563,A -85,B 0,C 180,E1 -15924.389,E2 -15924.389} C_VEL
LIN {X 0,Y 303.599,Z 399.791,A -85,B 0,C 180,E1 -15926.018,E2 -15926.018} C_VEL
LIN {X 0,Y 303.604,Z 400.379,A -85,B 0,C 180,E1 -15927.347,E2 -15927.347} C_VEL
LIN {X 0,Y 303.567,Z 400.548,A -85,B 0,C 180,E1 -15928.673,E2 -15928.673} C_VEL
LIN {X 0,Y 303.606,Z 400.308,A -85,B 0,C 180,E1 -15930,E2 -15930} C_VEL
LIN {X 0,Y 303.582,Z 399.679,A -85,B 0,C 180,E1 -15931.327,E2 -15931.327} C_VEL
LIN {X 0,Y 303.617,Z 398.66,A -85,B 0,C 180,E1 -15932.653,E2 -15932.653} C_VEL
LIN {X 0,Y 303.641,Z 397.206,A -85,B 0,C 180,E1 -15933.982,E2 -15933.982} C_VEL
LIN {X 0,Y 303.697,Z 394.711,A -85,B 0,C 180,E1 -15935.673,E2 -15935.673} C_VEL
LIN {X 0,Y 303.948,Z 390.13,A -85,B 0,C 180,E1 -15937.974,E2 -15937.974} C_VEL
LIN {X 0,Y 304.501,Z 383.854,A -85,B 0,C 180,E1 -15940.304,E2 -15940.304} C_VEL
LIN {X 0,Y 305.202,Z 377.005,A -85,B 0,C 180,E1 -15942.298,E2 -15942.298} C_VEL
LIN {X 0,Y 306.262,Z 368.468,A -85,B 0,C 180,E1 -15944.281,E2 -15944.281} C_VEL
LIN {X 0,Y 307.263,Z 359.652,A -85,B 0,C 180,E1 -15945.93,E2 -15945.93} C_VEL
LIN {X 0,Y 308.505,Z 348.79,A -85,B 0,C 180,E1 -15947.568,E2 -15947.568} C_VEL
LIN {X 0,Y 309.82,Z 337.941,A -85,B 0,C 180,E1 -15948.859,E2 -15948.859} C_VEL
LIN {X 0,Y 309.852,Z 333.045,A -85,B 0,C 180,E1 -15949.373,E2 -15949.373} C_VEL
LIN {X 0,Y 308.705,Z 321.146,A -85,B 0,C 180,E1 -15950.473,E2 -15950.473} C_VEL
LIN {X 0,Y 306.873,Z 307.601,A -85,B 0,C 180,E1 -15951.453,E2 -15951.453} C_VEL
LIN {X 0,Y 304.546,Z 294.107,A -85,B 0,C 180,E1 -15952.164,E2 -15952.164} C_VEL
LIN {X 0,Y 305.054,Z 288.316,A -85,B 0,C 180,E1 -15956.035,E2 -15956.035} C_VEL
LIN {X 0,Y 305.759,Z 281.952,A -85,B 0,C 180,E1 -15960.376,E2 -15960.376} C_VEL
LIN {X 0,Y 306.538,Z 276.243,A -85,B 0,C 180,E1 -15964.372,E2 -15964.372} C_VEL
LIN {X 0,Y 306.715,Z 273.069,A -85,B 0,C 180,E1 -15966.678,E2 -15966.678} C_VEL
LIN {X 0,Y 306.072,Z 268.784,A -85,B 0,C 180,E1 -15970.01,E2 -15970.01} C_VEL
LIN {X 0,Y 305.498,Z 265.432,A -85,B 0,C 180,E1 -15972.842,E2 -15972.842} C_VEL
LIN {X 0,Y 305.41,Z 265.442,A -85,B 0,C 180,E1 -15977.422,E2 -15977.422} C_VEL
LIN {X 0,Y 305.425,Z 265.439,A -85,B 0,C 180,E1 -15981.588,E2 -15981.588} C_VEL
LIN {X 0,Y 305.459,Z 265.437,A -85,B 0,C 180,E1 -15984.885,E2 -15984.885} C_VEL
LIN {X 0,Y 305.439,Z 265.438,A -85,B 0,C 180,E1 -15988.357,E2 -15988.357} C_VEL
LIN {X 0,Y 305.472,Z 265.432,A -85,B 0,C 180,E1 -15991.107,E2 -15991.107} C_VEL
LIN {X 0,Y 305.497,Z 265.43,A -85,B 0,C 180,E1 -15994.08,E2 -15994.08} C_VEL
LIN {X 0,Y 305.468,Z 265.437,A -85,B 0,C 180,E1 -15998.399,E2 -15998.399} C_VEL
LIN {X 0,Y 305.575,Z 265.418,A -85,B 0,C 180,E1 -16001.215,E2 -16001.215} C_VEL
LIN {X 0,Y 305.644,Z 265.41,A -85,B 0,C 180,E1 -16005.347,E2 -16005.347} C_VEL
LIN {X 0,Y 305.63,Z 265.411,A -85,B 0,C 180,E1 -16009.398,E2 -16009.398} C_VEL
LIN {X 0,Y 305.792,Z 265.397,A -85,B 0,C 180,E1 -16012.072,E2 -16012.072} C_VEL
LIN {X 0,Y 305.679,Z 265.405,A -85,B 0,C 180,E1 -16014.722,E2 -16014.722} C_VEL
LIN {X 0,Y 305.952,Z 265.365,A -85,B 0,C 180,E1 -16018.682,E2 -16018.682} C_VEL
LIN {X 0,Y 305.952,Z 265.368,A -85,B 0,C 180,E1 -16021.315,E2 -16021.315} C_VEL
LIN {X 0,Y 305.845,Z 265.385,A -85,B 0,C 180,E1 -16026.596,E2 -16026.596} C_VEL
LIN {X 0,Y 305.728,Z 265.4,A -85,B 0,C 180,E1 -16029.258,E2 -16029.258} C_VEL
LIN {X 0,Y 305.58,Z 265.421,A -85,B 0,C 180,E1 -16033.295,E2 -16033.295} C_VEL
LIN {X 0,Y 305.585,Z 265.417,A -85,B 0,C 180,E1 -16036.019,E2 -16036.019} C_VEL
LIN {X 0,Y 305.568,Z 265.424,A -85,B 0,C 180,E1 -16039.444,E2 -16039.444} C_VEL
LIN {X 0,Y 305.481,Z 265.432,A -85,B 0,C 180,E1 -16043.04,E2 -16043.04} C_VEL
LIN {X 0,Y 305.538,Z 265.423,A -85,B 0,C 180,E1 -16046.226,E2 -16046.226} C_VEL
LIN {X 0,Y 305.486,Z 265.433,A -85,B 0,C 180,E1 -16049.049,E2 -16049.049} C_VEL
LIN {X 0,Y 305.455,Z 265.435,A -85,B 0,C 180,E1 -16053.516,E2 -16053.516} C_VEL
LIN {X 0,Y 305.487,Z 265.431,A -85,B 0,C 180,E1 -16056.735,E2 -16056.735} C_VEL
LIN {X 0,Y 305.474,Z 265.433,A -85,B 0,C 180,E1 -16060.606,E2 -16060.606} C_VEL
LIN {X 0,Y 305.479,Z 265.43,A -85,B 0,C 180,E1 -16063.643,E2 -16063.643} C_VEL
LIN {X 0,Y 305.452,Z 265.433,A -85,B 0,C 180,E1 -16067.412,E2 -16067.412} C_VEL
LIN {X 0,Y 305.465,Z 265.432,A -85,B 0,C 180,E1 -16071.597,E2 -16071.597} C_VEL
LIN {X 0,Y 305.452,Z 265.437,A -85,B 0,C 180,E1 -16074.886,E2 -16074.886} C_VEL
LIN {X 0,Y 305.438,Z 265.44,A -85,B 0,C 180,E1 -16078.355,E2 -16078.355} C_VEL
LIN {X 0,Y 305.499,Z 265.429,A -85,B 0,C 180,E1 -16081.112,E2 -16081.112} C_VEL
LIN {X 0,Y 305.517,Z 265.429,A -85,B 0,C 180,E1 -16084.084,E2 -16084.084} C_VEL
LIN {X 0,Y 305.334,Z 265.627,A -85,B 0,C 180,E1 -16088.214,E2 -16088.214} C_VEL
LIN {X 0,Y 305.173,Z 268.627,A -85,B 0,C 180,E1 -16091.191,E2 -16091.191} C_VEL
LIN {X 0,Y 304.877,Z 273.105,A -85,B 0,C 180,E1 -16095.499,E2 -16095.499} C_VEL
LIN {X 0,Y 304.602,Z 277.273,A -85,B 0,C 180,E1 -16099.363,E2 -16099.363} C_VEL
LIN {X 0,Y 304.579,Z 279.103,A -85,B 0,C 180,E1 -16100.946,E2 -16100.946} C_VEL
LIN {X 0,Y 307.696,Z 292.464,A -85,B 0,C 180,E1 -16101.731,E2 -16101.731} C_VEL
LIN {X 0,Y 309.955,Z 305.392,A -85,B 0,C 180,E1 -16102.723,E2 -16102.723} C_VEL
LIN {X 0,Y 310.962,Z 313.818,A -85,B 0,C 180,E1 -16103.512,E2 -16103.512} C_VEL
LIN {X 0,Y 309.986,Z 324.756,A -85,B 0,C 180,E1 -16104.634,E2 -16104.634} C_VEL
LIN {X 0,Y 308.667,Z 335.981,A -85,B 0,C 180,E1 -16106.083,E2 -16106.083} C_VEL
LIN {X 0,Y 307.462,Z 345.908,A -85,B 0,C 180,E1 -16107.707,E2 -16107.707} C_VEL
LIN {X 0,Y 306.275,Z 355.534,A -85,B 0,C 180,E1 -16109.671,E2 -16109.671} C_VEL
LIN {X 0,Y 305.218,Z 363.215,A -85,B 0,C 180,E1 -16111.649,E2 -16111.649} C_VEL
LIN {X 0,Y 304.701,Z 368.457,A -85,B 0,C 180,E1 -16113.306,E2 -16113.306} C_VEL
LIN {X 0,Y 304.251,Z 373.537,A -85,B 0,C 180,E1 -16115.301,E2 -16115.301} C_VEL
LIN {X 0,Y 303.888,Z 377.493,A -85,B 0,C 180,E1 -16117.307,E2 -16117.307} C_VEL
LIN {X 0,Y 303.563,Z 380.419,A -85,B 0,C 180,E1 -16119.326,E2 -16119.326} C_VEL
LIN {X 0,Y 303.442,Z 381.801,A -85,B 0,C 180,E1 -16120.678,E2 -16120.678} C_VEL
LIN {X 0,Y 303.446,Z 382.78,A -85,B 0,C 180,E1 -16122.031,E2 -16122.031} C_VEL
LIN {X 0,Y 303.48,Z 383.382,A -85,B 0,C 180,E1 -16123.443,E2 -16123.443} C_VEL
LIN {X 0,Y 303.461,Z 383.511,A -85,B 0,C 180,E1 -16124.759,E2 -16124.759} C_VEL
LIN {X 0,Y 303.548,Z 383.238,A -85,B 0,C 180,E1 -16126.131,E2 -16126.131} C_VEL
LIN {X 0,Y 303.946,Z 381.75,A -85,B 0,C 180,E1 -16128.561,E2 -16128.561} C_VEL
LIN {X 0,Y 304.564,Z 378.963,A -85,B 0,C 180,E1 -16130.957,E2 -16130.957} C_VEL
LIN {X 0,Y 305.36,Z 375.381,A -85,B 0,C 180,E1 -16133.032,E2 -16133.032} C_VEL
LIN {X 0,Y 306.398,Z 370.598,A -85,B 0,C 180,E1 -16135.108,E2 -16135.108} C_VEL
LIN {X 0,Y 307.791,Z 364.464,A -85,B 0,C 180,E1 -16137.172,E2 -16137.172} C_VEL
LIN {X 0,Y 309.5,Z 356.751,A -85,B 0,C 180,E1 -16139.222,E2 -16139.222} C_VEL
LIN {X 0,Y 311.25,Z 348.146,A -85,B 0,C 180,E1 -16141.048,E2 -16141.048} C_VEL
LIN {X 0,Y 313.248,Z 337.881,A -85,B 0,C 180,E1 -16142.769,E2 -16142.769} C_VEL
LIN {X 0,Y 314.953,Z 327.868,A -85,B 0,C 180,E1 -16144.117,E2 -16144.117} C_VEL
LIN {X 0,Y 316.096,Z 320.893,A -85,B 0,C 180,E1 -16144.889,E2 -16144.889} C_VEL
LIN {X 0,Y 315.004,Z 312.996,A -85,B 0,C 180,E1 -16145.843,E2 -16145.843} C_VEL
LIN {X 0,Y 312.551,Z 302.167,A -85,B 0,C 180,E1 -16147.041,E2 -16147.041} C_VEL
LIN {X 0,Y 308.766,Z 289.811,A -85,B 0,C 180,E1 -16148.248,E2 -16148.248} C_VEL
LIN {X 0,Y 305.16,Z 280.155,A -85,B 0,C 180,E1 -16149.093,E2 -16149.093} C_VEL
LIN {X 0,Y 305.081,Z 279.586,A -85,B 0,C 180,E1 -16149.131,E2 -16149.131} C_VEL
LIN {X 0,Y 305.398,Z 276.242,A -85,B 0,C 180,E1 -16152.577,E2 -16152.577} C_VEL
LIN {X 0,Y 305.858,Z 272.684,A -85,B 0,C 180,E1 -16156.425,E2 -16156.425} C_VEL
LIN {X 0,Y 305.903,Z 269.603,A -85,B 0,C 180,E1 -16159.965,E2 -16159.965} C_VEL
LIN {X 0,Y 305.616,Z 266.693,A -85,B 0,C 180,E1 -16163.595,E2 -16163.595} C_VEL
LIN {X 0,Y 305.49,Z 265.708,A -85,B 0,C 180,E1 -16164.893,E2 -16164.893} C_VEL
LIN {X 0,Y 305.433,Z 265.443,A -85,B 0,C 180,E1 -16168.049,E2 -16168.049} C_VEL
LIN {X 0,Y 305.51,Z 265.43,A -85,B 0,C 180,E1 -16171.115,E2 -16171.115} C_VEL
LIN {X 0,Y 305.562,Z 265.424,A -85,B 0,C 180,E1 -16174.089,E2 -16174.089} C_VEL
LIN {X 0,Y 305.525,Z 265.429,A -85,B 0,C 180,E1 -16178.407,E2 -16178.407} C_VEL
LIN {X 0,Y 305.584,Z 265.421,A -85,B 0,C 180,E1 -16181.219,E2 -16181.219} C_VEL
LIN {X 0,Y 305.64,Z 265.409,A -85,B 0,C 180,E1 -16185.35,E2 -16185.35} C_VEL
LIN {X 0,Y 305.585,Z 265.415,A -85,B 0,C 180,E1 -16186.118,E2 -16186.118} C_VEL
LIN {X 0,Y 304.92,Z 265.504,A -85,B 0,C 180,E1 -16187.218,E2 -16187.218} C_VEL
LIN {X 0,Y 302.156,Z 265.854,A -85,B 0,C 180,E1 -16189.01,E2 -16189.01} C_VEL
LIN {X 0,Y 299.821,Z 266.145,A -85,B 0,C 180,E1 -16190.464,E2 -16190.464} C_VEL
LIN {X 0,Y 298.815,Z 266.265,A -85,B 0,C 180,E1 -16191.588,E2 -16191.588} C_VEL
LIN {X 0,Y 298.73,Z 266.273,A -85,B 0,C 180,E1 -16191.968,E2 -16191.968} C_VEL
LIN {X 0,Y 298.649,Z 266.286,A -85,B 0,C 180,E1 -16194.6,E2 -16194.6} C_VEL
LIN {X 0,Y 298.916,Z 266.252,A -85,B 0,C 180,E1 -16198.654,E2 -16198.654} C_VEL
LIN {X 0,Y 298.914,Z 266.251,A -85,B 0,C 180,E1 -16201.349,E2 -16201.349} C_VEL
LIN {X 0,Y 298.79,Z 266.268,A -85,B 0,C 180,E1 -16206.756,E2 -16206.756} C_VEL
LIN {X 0,Y 298.675,Z 266.281,A -85,B 0,C 180,E1 -16209.482,E2 -16209.482} C_VEL
LIN {X 0,Y 298.547,Z 266.297,A -85,B 0,C 180,E1 -16213.617,E2 -16213.617} C_VEL
LIN {X 0,Y 298.544,Z 266.301,A -85,B 0,C 180,E1 -16216.41,E2 -16216.41} C_VEL
LIN {X 0,Y 298.508,Z 266.306,A -85,B 0,C 180,E1 -16219.656,E2 -16219.656} C_VEL
LIN {X 0,Y 298.423,Z 266.319,A -85,B 0,C 180,E1 -16223.602,E2 -16223.602} C_VEL
LIN {X 0,Y 298.45,Z 266.316,A -85,B 0,C 180,E1 -16226.58,E2 -16226.58} C_VEL
LIN {X 0,Y 298.398,Z 266.32,A -85,B 0,C 180,E1 -16229.645,E2 -16229.645} C_VEL
LIN {X 0,Y 298.391,Z 266.319,A -85,B 0,C 180,E1 -16232.802,E2 -16232.802} C_VEL
LIN {X 0,Y 298.445,Z 266.311,A -85,B 0,C 180,E1 -16236.809,E2 -16236.809} C_VEL
LIN {X 0,Y 298.446,Z 266.37,A -85,B 0,C 180,E1 -16239.181,E2 -16239.181} C_VEL
LIN {X 0,Y 298.994,Z 269.993,A -85,B 0,C 180,E1 -16243.226,E2 -16243.226} C_VEL
LIN {X 0,Y 299.676,Z 273.816,A -85,B 0,C 180,E1 -16247.149,E2 -16247.149} C_VEL
LIN {X 0,Y 300.248,Z 277.718,A -85,B 0,C 180,E1 -16250.804,E2 -16250.804} C_VEL
LIN {X 0,Y 300.473,Z 279.839,A -85,B 0,C 180,E1 -16252.681,E2 -16252.681} C_VEL
LIN {X 0,Y 300.215,Z 283.667,A -85,B 0,C 180,E1 -16255.818,E2 -16255.818} C_VEL
LIN {X 0,Y 299.52,Z 287.653,A -85,B 0,C 180,E1 -16258.922,E2 -16258.922} C_VEL
LIN {X 0,Y 298.641,Z 293.323,A -85,B 0,C 180,E1 -16263.172,E2 -16263.172} C_VEL
LIN {X 0,Y 299.572,Z 296.65,A -85,B 0,C 180,E1 -16263.413,E2 -16263.413} C_VEL
LIN {X 0,Y 303.303,Z 309.161,A -85,B 0,C 180,E1 -16264.484,E2 -16264.484} C_VEL
LIN {X 0,Y 305.967,Z 321.506,A -85,B 0,C 180,E1 -16265.683,E2 -16265.683} C_VEL
LIN {X 0,Y 307.575,Z 332.709,A -85,B 0,C 180,E1 -16266.932,E2 -16266.932} C_VEL
LIN {X 0,Y 307.975,Z 341.762,A -85,B 0,C 180,E1 -16268.058,E2 -16268.058} C_VEL
LIN {X 0,Y 305.963,Z 352.739,A -85,B 0,C 180,E1 -16269.495,E2 -16269.495} C_VEL
LIN {X 0,Y 303.85,Z 362.554,A -85,B 0,C 180,E1 -16271.107,E2 -16271.107} C_VEL
LIN {X 0,Y 302.213,Z 370.614,A -85,B 0,C 180,E1 -16272.753,E2 -16272.753} C_VEL
LIN {X 0,Y 300.551,Z 378.552,A -85,B 0,C 180,E1 -16274.748,E2 -16274.748} C_VEL
LIN {X 0,Y 299.241,Z 383.95,A -85,B 0,C 180,E1 -16276.417,E2 -16276.417} C_VEL
LIN {X 0,Y 298.151,Z 389.255,A -85,B 0,C 180,E1 -16278.442,E2 -16278.442} C_VEL
LIN {X 0,Y 297.372,Z 393.41,A -85,B 0,C 180,E1 -16280.478,E2 -16280.478} C_VEL
LIN {X 0,Y 296.984,Z 395.624,A -85,B 0,C 180,E1 -16281.837,E2 -16281.837} C_VEL
LIN {X 0,Y 296.557,Z 398.699,A -85,B 0,C 180,E1 -16284.561,E2 -16284.561} C_VEL
LIN {X 0,Y 296.529,Z 400.208,A -85,B 0,C 180,E1 -16287.283,E2 -16287.283} C_VEL
LIN {X 0,Y 296.487,Z 400.336,A -85,B 0,C 180,E1 -16288.642,E2 -16288.642} C_VEL
LIN {X 0,Y 296.521,Z 400.073,A -85,B 0,C 180,E1 -16290,E2 -16290} C_VEL
LIN {X 0,Y 296.501,Z 399.422,A -85,B 0,C 180,E1 -16291.358,E2 -16291.358} C_VEL
LIN {X 0,Y 296.543,Z 398.378,A -85,B 0,C 180,E1 -16292.717,E2 -16292.717} C_VEL
LIN {X 0,Y 296.54,Z 396.877,A -85,B 0,C 180,E1 -16294.077,E2 -16294.077} C_VEL
LIN {X 0,Y 296.63,Z 393.825,A -85,B 0,C 180,E1 -16296.12,E2 -16296.12} C_VEL
LIN {X 0,Y 296.883,Z 389.697,A -85,B 0,C 180,E1 -16298.166,E2 -16298.166} C_VEL
LIN {X 0,Y 297.489,Z 383.363,A -85,B 0,C 180,E1 -16300.55,E2 -16300.55} C_VEL
LIN {X 0,Y 298.229,Z 376.449,A -85,B 0,C 180,E1 -16302.59,E2 -16302.59} C_VEL
LIN {X 0,Y 299.177,Z 369.388,A -85,B 0,C 180,E1 -16304.279,E2 -16304.279} C_VEL
LIN {X 0,Y 300.206,Z 360.855,A -85,B 0,C 180,E1 -16305.966,E2 -16305.966} C_VEL
LIN {X 0,Y 301.421,Z 350.284,A -85,B 0,C 180,E1 -16307.644,E2 -16307.644} C_VEL
LIN {X 0,Y 302.677,Z 339.825,A -85,B 0,C 180,E1 -16308.97,E2 -16308.97} C_VEL
LIN {X 0,Y 303.048,Z 335.202,A -85,B 0,C 180,E1 -16309.473,E2 -16309.473} C_VEL
LIN {X 0,Y 301.999,Z 323.676,A -85,B 0,C 180,E1 -16310.627,E2 -16310.627} C_VEL
LIN {X 0,Y 300.377,Z 310.544,A -85,B 0,C 180,E1 -16311.656,E2 -16311.656} C_VEL
LIN {X 0,Y 298.084,Z 297.211,A -85,B 0,C 180,E1 -16312.441,E2 -16312.441} C_VEL
LIN {X 0,Y 297.526,Z 293.86,A -85,B 0,C 180,E1 -16312.639,E2 -16312.639} C_VEL
LIN {X 0,Y 298.068,Z 288.076,A -85,B 0,C 180,E1 -16316.614,E2 -16316.614} C_VEL
LIN {X 0,Y 298.863,Z 281.593,A -85,B 0,C 180,E1 -16321.154,E2 -16321.154} C_VEL
LIN {X 0,Y 299.58,Z 276.533,A -85,B 0,C 180,E1 -16324.805,E2 -16324.805} C_VEL
LIN {X 0,Y 299.602,Z 272.875,A -85,B 0,C 180,E1 -16327.581,E2 -16327.581} C_VEL
LIN {X 0,Y 298.793,Z 268.406,A -85,B 0,C 180,E1 -16331.192,E2 -16331.192} C_VEL
LIN {X 0,Y 298.428,Z 266.314,A -85,B 0,C 180,E1 -16333.107,E2 -16333.107} C_VEL
LIN {X 0,Y 298.368,Z 266.323,A -85,B 0,C 180,E1 -16336.913,E2 -16336.913} C_VEL
LIN {X 0,Y 298.383,Z 266.319,A -85,B 0,C 180,E1 -16341.01,E2 -16341.01} C_VEL
LIN {X 0,Y 298.402,Z 266.313,A -85,B 0,C 180,E1 -16343.926,E2 -16343.926} C_VEL
LIN {X 0,Y 298.391,Z 266.315,A -85,B 0,C 180,E1 -16347.198,E2 -16347.198} C_VEL
LIN {X 0,Y 298.399,Z 266.316,A -85,B 0,C 180,E1 -16350.624,E2 -16350.624} C_VEL
LIN {X 0,Y 298.436,Z 266.309,A -85,B 0,C 180,E1 -16354.918,E2 -16354.918} C_VEL
LIN {X 0,Y 298.402,Z 266.313,A -85,B 0,C 180,E1 -16357.861,E2 -16357.861} C_VEL
LIN {X 0,Y 298.521,Z 266.299,A -85,B 0,C 180,E1 -16360.754,E2 -16360.754} C_VEL
LIN {X 0,Y 298.589,Z 266.29,A -85,B 0,C 180,E1 -16364.993,E2 -16364.993} C_VEL
LIN {X 0,Y 298.586,Z 266.288,A -85,B 0,C 180,E1 -16369.145,E2 -16369.145} C_VEL
LIN {X 0,Y 298.736,Z 266.274,A -85,B 0,C 180,E1 -16371.884,E2 -16371.884} C_VEL
LIN {X 0,Y 298.65,Z 266.281,A -85,B 0,C 180,E1 -16374.597,E2 -16374.597} C_VEL
